C05482=1238.622,-59.773,-37.360,-179.966,5.213,148.890
C05483=1238.616,-59.523,-37.372,-179.963,5.213,148.889
C05484=1238.612,-59.273,-37.385,-179.961,5.213,148.889
C05485=1238.607,-59.024,-37.398,-179.958,5.213,148.888
C05486=1238.602,-58.774,-37.409,-179.956,5.214,148.887
C05487=1238.597,-58.525,-37.422,-179.953,5.214,148.887
C05488=1238.591,-58.275,-37.433,-179.951,5.214,148.886
C05489=1238.586,-58.026,-37.446,-179.949,5.214,148.885
C05490=1238.581,-57.777,-37.459,-179.946,5.214,148.884
C05491=1238.576,-57.526,-37.471,-179.943,5.214,148.884
C05492=1238.571,-57.277,-37.484,-179.941,5.214,148.883
C05493=1238.566,-57.027,-37.496,-179.939,5.214,148.882
C05494=1238.561,-56.777,-37.508,-179.936,5.214,148.881
C05495=1238.555,-56.528,-37.521,-179.934,5.214,148.881
C05496=1238.550,-56.279,-37.533,-179.931,5.214,148.880
C05497=1238.545,-56.028,-37.545,-179.929,5.214,148.879
C05498=1238.540,-55.779,-37.558,-179.927,5.215,148.879
C05499=1238.535,-55.529,-37.571,-179.924,5.214,148.878
C05500=1238.530,-55.280,-37.583,-179.922,5.215,148.877
C05501=1238.525,-55.030,-37.595,-179.920,5.214,148.877
C05502=1238.520,-54.780,-37.608,-179.917,5.215,148.876
C05503=1238.515,-54.530,-37.620,-179.914,5.215,148.875
C05504=1238.510,-54.281,-37.633,-179.912,5.215,148.874
C05505=1238.504,-54.032,-37.645,-179.909,5.215,148.873
C05506=1238.499,-53.782,-37.658,-179.907,5.215,148.873
C05507=1238.495,-53.532,-37.670,-179.904,5.215,148.872
C05508=1238.489,-53.282,-37.683,-179.902,5.215,148.871
C05509=1238.484,-53.033,-37.695,-179.900,5.216,148.871
C05510=1238.478,-52.783,-37.708,-179.898,5.215,148.870
C05511=1238.473,-52.533,-37.720,-179.895,5.216,148.869
C05512=1238.468,-52.283,-37.733,-179.893,5.215,148.869
C05513=1238.463,-52.034,-37.746,-179.890,5.216,148.868
C05514=1238.458,-51.785,-37.759,-179.888,5.216,148.867
C05515=1238.453,-51.536,-37.771,-179.885,5.216,148.866
C05516=1238.448,-51.285,-37.783,-179.882,5.216,148.865
C05517=1238.443,-51.036,-37.796,-179.880,5.216,148.865
C05518=1238.438,-50.786,-37.809,-179.877,5.216,148.864
C05519=1238.433,-50.537,-37.821,-179.875,5.216,148.863
C05520=1238.428,-50.287,-37.834,-179.873,5.217,148.863
C05521=1238.422,-50.037,-37.847,-179.871,5.216,148.862
C05522=1238.417,-49.788,-37.860,-179.868,5.217,148.861
C05523=1238.412,-49.538,-37.872,-179.866,5.216,148.861
C05524=1238.407,-49.288,-37.885,-179.863,5.217,148.860
C05525=1238.402,-49.039,-37.897,-179.861,5.217,148.859
C05526=1238.397,-48.789,-37.910,-179.858,5.217,148.858
C05527=1238.391,-48.519,-37.924,-179.855,5.217,148.858
C05528=1238.386,-48.250,-37.938,-179.853,5.217,148.857
C05529=1238.381,-47.981,-37.951,-179.850,5.217,148.856
C05530=1238.375,-47.711,-37.966,-179.847,5.217,148.855
C05531=1238.370,-47.461,-37.978,-179.845,5.217,148.854
C05532=1238.365,-47.212,-37.991,-179.843,5.218,148.854
C05533=1238.360,-46.962,-38.004,-179.840,5.217,148.853
C05534=1238.354,-46.712,-38.016,-179.838,5.218,148.852
C05535=1238.349,-46.462,-38.029,-179.836,5.218,148.852
C05536=1238.345,-46.212,-38.042,-179.833,5.218,148.851
C05537=1238.339,-45.963,-38.054,-179.830,5.219,148.850
C05538=1238.334,-45.714,-38.067,-179.828,5.218,148.850
C05539=1238.329,-45.463,-38.081,-179.826,5.219,148.849
C05540=1238.324,-45.214,-38.093,-179.823,5.218,148.848
C05541=1238.319,-44.965,-38.106,-179.820,5.219,148.847
C05542=1238.314,-44.715,-38.119,-179.818,5.218,148.847
C05543=1238.308,-44.465,-38.132,-179.816,5.219,148.846
C05544=1238.303,-44.216,-38.144,-179.814,5.218,148.845
C05545=1238.298,-43.966,-38.157,-179.811,5.219,148.844
C05546=1238.294,-43.716,-38.170,-179.808,5.219,148.844
C05547=1238.288,-43.467,-38.183,-179.806,5.219,148.843
C05548=1238.283,-43.217,-38.196,-179.803,5.220,148.842
C05549=1238.278,-42.967,-38.209,-179.801,5.219,148.842
C05550=1238.273,-42.719,-38.222,-179.799,5.220,148.841
C05551=1238.268,-42.468,-38.236,-179.796,5.219,148.840
C05552=1238.263,-42.219,-38.248,-179.793,5.220,148.839
C05553=1238.258,-41.970,-38.261,-179.791,5.219,148.839
C05554=1238.252,-41.719,-38.274,-179.789,5.220,148.838
C05555=1238.247,-41.470,-38.287,-179.786,5.220,148.837
C05556=1238.242,-41.221,-38.300,-179.784,5.220,148.836
C05557=1238.238,-40.971,-38.313,-179.781,5.220,148.836
C05558=1238.232,-40.721,-38.326,-179.779,5.220,148.835
C05559=1238.227,-40.471,-38.339,-179.777,5.221,148.834
C05560=1238.223,-40.222,-38.352,-179.774,5.220,148.834
C05561=1238.217,-39.973,-38.365,-179.772,5.221,148.833
C05562=1238.212,-39.723,-38.378,-179.769,5.221,148.832
C05563=1238.207,-39.473,-38.391,-179.767,5.221,148.831
C05564=1238.202,-39.223,-38.404,-179.764,5.221,148.831
C05565=1238.197,-38.974,-38.417,-179.762,5.221,148.830
C05566=1238.192,-38.725,-38.430,-179.759,5.221,148.829
C05567=1238.187,-38.475,-38.444,-179.757,5.221,148.829
C05568=1238.181,-38.225,-38.457,-179.754,5.222,148.828
C05569=1238.176,-37.975,-38.470,-179.752,5.222,148.827
C05570=1238.171,-37.726,-38.483,-179.750,5.222,148.826
C05571=1238.166,-37.477,-38.495,-179.747,5.222,148.826
C05572=1238.161,-37.227,-38.510,-179.745,5.222,148.825
C05573=1238.156,-36.977,-38.522,-179.742,5.222,148.824
C05574=1238.151,-36.727,-38.536,-179.740,5.222,148.824
C05575=1238.145,-36.478,-38.548,-179.737,5.222,148.823
C05576=1238.141,-36.228,-38.562,-179.734,5.223,148.822
C05577=1238.135,-35.979,-38.575,-179.732,5.222,148.821
C05578=1238.130,-35.729,-38.588,-179.730,5.223,148.821
C05579=1238.125,-35.479,-38.601,-179.728,5.223,148.820
C05580=1238.120,-35.230,-38.615,-179.725,5.223,148.819
C05581=1238.115,-34.980,-38.628,-179.722,5.224,148.819
C05582=1238.110,-34.731,-38.641,-179.720,5.223,148.818
C05583=1238.106,-34.481,-38.655,-179.717,5.224,148.817
C05584=1238.100,-34.232,-38.668,-179.715,5.224,148.816
C05585=1238.095,-33.982,-38.681,-179.713,5.224,148.816
C05586=1238.090,-33.733,-38.695,-179.711,5.224,148.815
C05587=1238.085,-33.483,-38.708,-179.707,5.224,148.814
C05588=1238.079,-33.233,-38.721,-179.705,5.224,148.813
C05589=1238.075,-32.984,-38.734,-179.703,5.224,148.813
C05590=1238.069,-32.734,-38.748,-179.700,5.225,148.812
C05591=1238.065,-32.484,-38.761,-179.698,5.224,148.811
C05592=1238.059,-32.235,-38.775,-179.695,5.225,148.811
C05593=1238.055,-31.985,-38.787,-179.693,5.225,148.810
C05594=1238.049,-31.735,-38.801,-179.691,5.225,148.809
C05595=1238.044,-31.486,-38.814,-179.688,5.226,148.809
C05596=1238.039,-31.236,-38.828,-179.686,5.225,148.808
C05597=1238.034,-30.987,-38.841,-179.683,5.226,148.807
C05598=1238.029,-30.737,-38.854,-179.681,5.225,148.806
C05599=1238.024,-30.487,-38.867,-179.678,5.226,148.805
C05600=1238.018,-30.238,-38.881,-179.675,5.226,148.805
C05601=1238.014,-29.988,-38.894,-179.673,5.226,148.804
C05602=1238.008,-29.739,-38.908,-179.671,5.226,148.803
C05603=1238.004,-29.489,-38.921,-179.668,5.226,148.803
C05604=1237.998,-29.240,-38.935,-179.666,5.227,148.802
C05605=1237.993,-28.990,-38.949,-179.663,5.227,148.801
C05606=1237.988,-28.741,-38.962,-179.661,5.227,148.801
C05607=1237.983,-28.491,-38.975,-179.658,5.227,148.800
C05608=1237.978,-28.242,-38.988,-179.656,5.227,148.799
C05609=1237.973,-27.992,-39.002,-179.654,5.227,148.798
C05610=1237.968,-27.742,-39.015,-179.651,5.228,148.798
C05611=1237.963,-27.493,-39.029,-179.649,5.228,148.797
C05612=1237.958,-27.243,-39.044,-179.646,5.228,148.796
C05613=1237.953,-26.994,-39.056,-179.644,5.228,148.795
C05614=1237.948,-26.744,-39.070,-179.641,5.228,148.795
C05615=1237.943,-26.495,-39.083,-179.638,5.229,148.794
C05616=1237.938,-26.245,-39.097,-179.636,5.228,148.793
C05617=1237.932,-25.995,-39.111,-179.634,5.229,148.793
C05618=1237.928,-25.746,-39.124,-179.631,5.228,148.792
C05619=1237.922,-25.496,-39.138,-179.629,5.229,148.791
C05620=1237.917,-25.247,-39.152,-179.626,5.229,148.791
C05621=1237.912,-24.997,-39.165,-179.624,5.229,148.790
C05622=1237.907,-24.747,-39.179,-179.621,5.230,148.789
C05623=1237.903,-24.498,-39.192,-179.619,5.229,148.789
C05624=1237.897,-24.248,-39.206,-179.616,5.230,148.788
C05625=1237.892,-23.999,-39.220,-179.614,5.230,148.787
C05626=1237.887,-23.749,-39.233,-179.611,5.230,148.786
C05627=1237.882,-23.499,-39.247,-179.609,5.230,148.785
C05628=1237.877,-23.250,-39.261,-179.606,5.231,148.785
C05629=1237.871,-23.000,-39.274,-179.604,5.230,148.784
C05630=1237.867,-22.750,-39.288,-179.601,5.231,148.783
C05631=1237.861,-22.482,-39.303,-179.599,5.232,148.783
C05632=1237.856,-22.212,-39.318,-179.596,5.231,148.782
C05633=1237.850,-21.943,-39.333,-179.593,5.231,148.781
C05634=1237.845,-21.674,-39.348,-179.591,5.232,148.780
C05635=1237.840,-21.425,-39.361,-179.589,5.232,148.780
C05636=1237.835,-21.174,-39.375,-179.586,5.232,148.779
C05637=1237.830,-20.925,-39.389,-179.583,5.232,148.778
C05638=1237.824,-20.676,-39.403,-179.581,5.232,148.777
C05639=1237.820,-20.426,-39.416,-179.578,5.232,148.777
C05640=1237.815,-20.176,-39.430,-179.576,5.232,148.776
C05641=1237.809,-19.927,-39.444,-179.573,5.233,148.775
C05642=1237.804,-19.677,-39.458,-179.571,5.233,148.775
C05643=1237.800,-19.427,-39.471,-179.569,5.233,148.774
C05644=1237.794,-19.178,-39.485,-179.566,5.233,148.773
C05645=1237.789,-18.929,-39.499,-179.563,5.234,148.773
C05646=1237.784,-18.679,-39.514,-179.561,5.234,148.772
C05647=1237.779,-18.430,-39.526,-179.559,5.234,148.771
C05648=1237.774,-18.180,-39.540,-179.557,5.234,148.770
C05649=1237.769,-17.930,-39.555,-179.554,5.234,148.770
C05650=1237.764,-17.681,-39.569,-179.551,5.235,148.769
C05651=1237.759,-17.431,-39.583,-179.549,5.234,148.768
C05652=1237.754,-17.181,-39.596,-179.546,5.235,148.767
C05653=1237.749,-16.932,-39.610,-179.543,5.235,148.767
C05654=1237.744,-16.683,-39.624,-179.541,5.235,148.766
C05655=1237.739,-16.433,-39.638,-179.539,5.236,148.765
C05656=1237.734,-16.183,-39.653,-179.537,5.235,148.765
C05657=1237.728,-15.934,-39.667,-179.534,5.236,148.764
C05658=1237.724,-15.685,-39.680,-179.531,5.236,148.763
C05659=1237.719,-15.435,-39.694,-179.529,5.236,148.763
C05660=1237.714,-15.185,-39.708,-179.526,5.237,148.762
C05661=1237.708,-14.936,-39.722,-179.524,5.237,148.761
C05662=1237.703,-14.686,-39.736,-179.522,5.237,148.760
C05663=1237.698,-14.436,-39.751,-179.519,5.237,148.760
C05664=1237.693,-14.187,-39.764,-179.516,5.237,148.759
C05665=1237.689,-13.938,-39.778,-179.514,5.237,148.758
C05666=1237.684,-13.688,-39.792,-179.511,5.238,148.757
C05667=1237.679,-13.439,-39.807,-179.509,5.237,148.757
C05668=1237.674,-13.189,-39.821,-179.506,5.238,148.756
C05669=1237.668,-12.939,-39.834,-179.504,5.238,148.755
C05670=1237.663,-12.689,-39.848,-179.502,5.238,148.755
C05671=1237.658,-12.440,-39.863,-179.499,5.239,148.754
C05672=1237.653,-12.190,-39.877,-179.496,5.239,148.753
C05673=1237.647,-11.941,-39.891,-179.494,5.239,148.753
C05674=1237.642,-11.691,-39.905,-179.492,5.239,148.752
C05675=1237.638,-11.442,-39.919,-179.489,5.240,148.751
C05676=1237.633,-11.192,-39.933,-179.487,5.240,148.751
C05677=1237.628,-10.943,-39.947,-179.484,5.240,148.750
C05678=1237.623,-10.694,-39.961,-179.482,5.241,148.749
C05679=1237.618,-10.444,-39.976,-179.479,5.240,148.748
C05680=1237.613,-10.194,-39.990,-179.476,5.241,148.748
C05681=1237.608,-9.944,-40.004,-179.474,5.241,148.747
C05682=1237.603,-9.695,-40.018,-179.472,5.241,148.746
C05683=1237.597,-9.446,-40.032,-179.469,5.241,148.745
C05684=1237.592,-9.196,-40.047,-179.467,5.241,148.745
C05685=1237.588,-8.947,-40.062,-179.464,5.242,148.744
C05686=1237.583,-8.697,-40.076,-179.462,5.242,148.743
C05687=1237.578,-8.447,-40.090,-179.460,5.242,148.743
C05688=1237.573,-8.198,-40.104,-179.457,5.242,148.742
C05689=1237.567,-7.949,-40.118,-179.454,5.243,148.741
C05690=1237.562,-7.699,-40.133,-179.452,5.243,148.741
C05691=1237.557,-7.449,-40.147,-179.449,5.243,148.740
C05692=1237.553,-7.200,-40.161,-179.447,5.244,148.739
C05693=1237.548,-6.950,-40.175,-179.445,5.243,148.739
C05694=1237.543,-6.700,-40.190,-179.442,5.244,148.738
C05695=1237.537,-6.452,-40.204,-179.439,5.244,148.737
C05696=1237.532,-6.202,-40.219,-179.437,5.244,148.736
C05697=1237.527,-5.952,-40.233,-179.434,5.244,148.736
C05698=1237.523,-5.703,-40.247,-179.432,5.245,148.735
C05699=1237.518,-5.453,-40.261,-179.429,5.245,148.734
C05700=1237.512,-5.203,-40.276,-179.427,5.245,148.733
C05701=1237.507,-4.954,-40.291,-179.424,5.246,148.733
C05702=1237.502,-4.704,-40.306,-179.422,5.245,148.732
C05703=1237.497,-4.455,-40.320,-179.419,5.246,148.731
C05704=1237.492,-4.205,-40.334,-179.417,5.246,148.731
C05705=1237.487,-3.956,-40.348,-179.415,5.246,148.730
C05706=1237.482,-3.707,-40.363,-179.412,5.247,148.729
C05707=1237.477,-3.457,-40.377,-179.409,5.247,148.729
C05708=1237.472,-3.207,-40.392,-179.407,5.247,148.728
C05709=1237.467,-2.957,-40.406,-179.405,5.247,148.727
C05710=1237.463,-2.708,-40.421,-179.402,5.248,148.727
C05711=1237.457,-2.458,-40.436,-179.399,5.247,148.726
C05712=1237.452,-2.209,-40.450,-179.397,5.248,148.725
C05713=1237.446,-1.960,-40.464,-179.394,5.248,148.724
C05714=1237.442,-1.711,-40.479,-179.392,5.248,148.724
C05715=1237.437,-1.461,-40.493,-179.389,5.249,148.723
C05716=1237.432,-1.211,-40.508,-179.387,5.249,148.722
C05717=1237.427,-0.961,-40.522,-179.385,5.249,148.721
C05718=1237.422,-0.712,-40.537,-179.382,5.249,148.721
C05719=1237.417,-0.462,-40.552,-179.379,5.250,148.720
C05720=1237.412,-0.213,-40.566,-179.377,5.251,148.719
C05721=1237.407,0.037,-40.581,-179.375,5.250,148.719
C05722=1237.402,0.286,-40.595,-179.372,5.251,148.718
C05723=1237.396,0.536,-40.610,-179.369,5.251,148.717
C05724=1237.392,0.785,-40.625,-179.367,5.251,148.717
C05725=1237.387,1.035,-40.639,-179.365,5.252,148.716
C05726=1237.382,1.284,-40.654,-179.362,5.252,148.715
C05727=1237.377,1.534,-40.669,-179.360,5.252,148.715
C05728=1237.371,1.784,-40.684,-179.357,5.252,148.714
C05729=1237.367,2.033,-40.698,-179.355,5.253,148.713
C05730=1237.362,2.283,-40.713,-179.352,5.252,148.712
C05731=1237.357,2.532,-40.728,-179.349,5.253,148.712
C05732=1237.351,2.782,-40.743,-179.347,5.253,148.711
C05733=1237.347,3.031,-40.757,-179.345,5.253,148.710
C05734=1237.342,3.281,-40.772,-179.342,5.254,148.710
C05735=1237.337,3.549,-40.788,-179.339,5.254,148.709
C05736=1237.330,3.818,-40.804,-179.337,5.255,148.708
C05737=1237.325,4.087,-40.819,-179.333,5.255,148.707
C05738=1237.320,4.355,-40.835,-179.331,5.255,148.707
C05739=1237.314,4.605,-40.850,-179.329,5.255,148.706
C05740=1237.310,4.854,-40.865,-179.326,5.256,148.705
C05741=1237.305,5.104,-40.879,-179.323,5.256,148.705
C05742=1237.299,5.354,-40.895,-179.321,5.256,148.704
C05743=1237.294,5.603,-40.909,-179.319,5.256,148.703
C05744=1237.290,5.853,-40.924,-179.316,5.257,148.702
C05745=1237.285,6.103,-40.939,-179.314,5.257,148.702
C05746=1237.280,6.352,-40.954,-179.311,5.257,148.701
C05747=1237.275,6.602,-40.968,-179.309,5.258,148.700
C05748=1237.270,6.851,-40.983,-179.307,5.258,148.700
C05749=1237.265,7.100,-40.999,-179.304,5.258,148.699
C05750=1237.260,7.350,-41.013,-179.301,5.259,148.698
C05751=1237.255,7.599,-41.028,-179.299,5.259,148.698
C05752=1237.250,7.849,-41.043,-179.297,5.259,148.697
C05753=1237.245,8.098,-41.058,-179.294,5.259,148.696
C05754=1237.240,8.348,-41.072,-179.291,5.260,148.695
C05755=1237.235,8.597,-41.088,-179.289,5.259,148.695
C05756=1237.230,8.847,-41.103,-179.286,5.260,148.694
C05757=1237.224,9.097,-41.118,-179.283,5.260,148.693
C05758=1237.220,9.346,-41.133,-179.281,5.261,148.693
C05759=1237.215,9.595,-41.148,-179.279,5.261,148.692
C05760=1237.209,9.845,-41.163,-179.276,5.261,148.691
C05761=1237.205,10.095,-41.178,-179.273,5.262,148.691
C05762=1237.200,10.345,-41.193,-179.271,5.262,148.690
C05763=1237.195,10.594,-41.208,-179.269,5.262,148.689
C05764=1237.190,10.843,-41.223,-179.266,5.263,148.688
C05765=1237.185,11.093,-41.238,-179.263,5.263,148.688
C05766=1237.180,11.342,-41.253,-179.261,5.263,148.687
C05767=1237.175,11.591,-41.268,-179.259,5.263,148.686
C05768=1237.170,11.840,-41.283,-179.256,5.264,148.686
C05769=1237.164,12.090,-41.298,-179.254,5.264,148.685
C05770=1237.160,12.340,-41.314,-179.251,5.264,148.684
C05771=1237.156,12.589,-41.329,-179.249,5.265,148.684
C05772=1237.150,12.839,-41.344,-179.246,5.265,148.683
C05773=1237.145,13.088,-41.359,-179.244,5.265,148.682
C05774=1237.140,13.338,-41.374,-179.241,5.266,148.682
C05775=1237.135,13.587,-41.389,-179.239,5.266,148.681
C05776=1237.130,13.837,-41.404,-179.236,5.267,148.680
C05777=1237.125,14.086,-41.419,-179.234,5.266,148.680
C05778=1237.120,14.336,-41.435,-179.231,5.267,148.679
C05779=1237.115,14.585,-41.450,-179.229,5.268,148.678
C05780=1237.110,14.835,-41.466,-179.226,5.267,148.678
C05781=1237.105,15.084,-41.480,-179.224,5.268,148.677
C05782=1237.100,15.334,-41.495,-179.221,5.268,148.676
C05783=1237.095,15.583,-41.510,-179.219,5.269,148.675
C05784=1237.090,15.833,-41.526,-179.216,5.269,148.675
C05785=1237.086,16.082,-41.541,-179.214,5.269,148.674
C05786=1237.080,16.332,-41.556,-179.211,5.270,148.673
C05787=1237.075,16.581,-41.571,-179.208,5.270,148.673
C05788=1237.070,16.830,-41.587,-179.206,5.270,148.672
C05789=1237.065,17.081,-41.603,-179.203,5.270,148.671
C05790=1237.060,17.330,-41.618,-179.201,5.271,148.670
C05791=1237.055,17.579,-41.633,-179.198,5.271,148.670
C05792=1237.050,17.828,-41.648,-179.196,5.271,148.669
C05793=1237.045,18.078,-41.664,-179.193,5.272,148.668
C05794=1237.041,18.328,-41.679,-179.191,5.272,148.668
C05795=1237.035,18.577,-41.694,-179.188,5.273,148.667
C05796=1237.030,18.827,-41.710,-179.186,5.272,148.666
C05797=1237.025,19.076,-41.725,-179.183,5.273,148.666
C05798=1237.020,19.325,-41.740,-179.181,5.274,148.665
C05799=1237.016,19.575,-41.756,-179.178,5.274,148.664
C05800=1237.010,19.824,-41.771,-179.176,5.274,148.664
C05801=1237.005,20.074,-41.787,-179.173,5.274,148.663
C05802=1237.000,20.323,-41.802,-179.171,5.275,148.662
C05803=1236.996,20.573,-41.818,-179.168,5.276,148.662
C05804=1236.990,20.822,-41.833,-179.166,5.275,148.661
C05805=1236.986,21.072,-41.848,-179.163,5.276,148.660
C05806=1236.980,21.321,-41.864,-179.161,5.276,148.660
C05807=1236.976,21.571,-41.879,-179.158,5.277,148.659
C05808=1236.971,21.820,-41.895,-179.156,5.277,148.658
C05809=1236.965,22.070,-41.910,-179.153,5.277,148.657
C05810=1236.961,22.319,-41.925,-179.151,5.278,148.657
C05811=1236.956,22.569,-41.941,-179.148,5.278,148.656
C05812=1236.951,22.818,-41.957,-179.146,5.278,148.655
C05813=1236.945,23.068,-41.973,-179.143,5.279,148.655
C05814=1236.941,23.317,-41.988,-179.141,5.279,148.654
C05815=1236.936,23.567,-42.004,-179.138,5.280,148.653
C05816=1236.930,23.816,-42.019,-179.136,5.279,148.653
C05817=1236.926,24.065,-42.034,-179.133,5.280,148.652
C05818=1236.921,24.315,-42.050,-179.131,5.281,148.651
C05819=1236.916,24.564,-42.066,-179.128,5.281,148.651
C05820=1236.911,24.813,-42.081,-179.125,5.282,148.650
C05821=1236.906,25.063,-42.097,-179.123,5.281,148.649
C05822=1236.901,25.313,-42.113,-179.121,5.282,148.649
C05823=1236.896,25.562,-42.128,-179.118,5.283,148.648
C05824=1236.891,25.811,-42.143,-179.115,5.283,148.647
C05825=1236.886,26.061,-42.159,-179.113,5.283,148.647
C05826=1236.881,26.311,-42.175,-179.111,5.283,148.646
C05827=1236.876,26.560,-42.191,-179.108,5.284,148.645
C05828=1236.872,26.809,-42.207,-179.105,5.285,148.645
C05829=1236.866,27.059,-42.222,-179.103,5.285,148.644
C05830=1236.861,27.308,-42.238,-179.100,5.285,148.643
C05831=1236.856,27.558,-42.254,-179.098,5.285,148.642
C05832=1236.851,27.807,-42.270,-179.095,5.286,148.642
C05833=1236.846,28.056,-42.285,-179.093,5.286,148.641
C05834=1236.842,28.306,-42.301,-179.090,5.286,148.640
C05835=1236.836,28.556,-42.317,-179.088,5.287,148.640
C05836=1236.831,28.806,-42.333,-179.085,5.287,148.639
C05837=1236.826,29.054,-42.349,-179.083,5.288,148.638
C05838=1236.822,29.304,-42.364,-179.080,5.288,148.638
C05839=1236.816,29.572,-42.381,-179.078,5.288,148.637
C05840=1236.811,29.841,-42.398,-179.075,5.289,148.636
C05841=1236.806,30.110,-42.415,-179.073,5.289,148.636
C05842=1236.800,30.378,-42.432,-179.069,5.290,148.635
C05843=1236.795,30.628,-42.448,-179.067,5.290,148.634
C05844=1236.790,30.877,-42.465,-179.064,5.291,148.633
C05845=1236.785,31.126,-42.480,-179.061,5.291,148.633
C05846=1236.781,31.376,-42.496,-179.059,5.291,148.632
C05847=1236.775,31.626,-42.511,-179.057,5.292,148.631
C05848=1236.771,31.875,-42.528,-179.054,5.292,148.631
C05849=1236.765,32.125,-42.543,-179.051,5.293,148.630
C05850=1236.760,32.374,-42.559,-179.049,5.293,148.629
C05851=1236.756,32.623,-42.576,-179.047,5.293,148.629
C05852=1236.750,32.873,-42.591,-179.045,5.294,148.628
C05853=1236.746,33.122,-42.608,-179.042,5.294,148.628
C05854=1236.740,33.372,-42.623,-179.039,5.295,148.627
C05855=1236.735,33.621,-42.639,-179.037,5.296,148.626
C05856=1236.731,33.870,-42.655,-179.035,5.295,148.626
C05857=1236.726,34.120,-42.671,-179.032,5.296,148.625
C05858=1236.721,34.369,-42.687,-179.029,5.296,148.624
C05859=1236.716,34.619,-42.703,-179.027,5.297,148.623
C05860=1236.711,34.869,-42.719,-179.024,5.298,148.623
C05861=1236.706,35.117,-42.735,-179.022,5.297,148.622
C05862=1236.701,35.368,-42.751,-179.019,5.298,148.621
C05863=1236.696,35.616,-42.768,-179.017,5.298,148.621
C05864=1236.691,35.866,-42.783,-179.014,5.299,148.620
C05865=1236.686,36.115,-42.800,-179.011,5.300,148.619
C05866=1236.681,36.365,-42.815,-179.009,5.300,148.619
C05867=1236.677,36.614,-42.832,-179.007,5.300,148.618
C05868=1236.671,36.864,-42.848,-179.004,5.300,148.617
C05869=1236.667,37.113,-42.864,-179.001,5.301,148.617
C05870=1236.661,37.362,-42.880,-178.999,5.302,148.616
C05871=1236.657,37.612,-42.897,-178.996,5.302,148.615
C05872=1236.651,37.861,-42.912,-178.994,5.302,148.615
C05873=1236.647,38.111,-42.929,-178.991,5.303,148.614
C05874=1236.642,38.360,-42.944,-178.989,5.303,148.613
C05875=1236.637,38.610,-42.961,-178.986,5.304,148.613
C05876=1236.632,38.859,-42.977,-178.983,5.304,148.612
C05877=1236.627,39.109,-42.993,-178.981,5.305,148.611
C05878=1236.622,39.358,-43.009,-178.979,5.305,148.611
C05879=1236.617,39.607,-43.026,-178.976,5.305,148.610
C05880=1236.612,39.856,-43.042,-178.974,5.306,148.609
C05881=1236.607,40.107,-43.058,-178.971,5.306,148.609
C05882=1236.602,40.355,-43.075,-178.968,5.307,148.608
C05883=1236.597,40.606,-43.091,-178.966,5.307,148.607
C05884=1236.592,40.854,-43.107,-178.964,5.307,148.607
C05885=1236.587,41.104,-43.124,-178.961,5.308,148.606
C05886=1236.583,41.354,-43.140,-178.959,5.309,148.605
C05887=1236.577,41.603,-43.156,-178.956,5.309,148.605
C05888=1236.573,41.852,-43.173,-178.953,5.310,148.604
C05889=1236.568,42.102,-43.188,-178.951,5.310,148.603
C05890=1236.563,42.351,-43.205,-178.949,5.310,148.603
C05891=1236.557,42.600,-43.222,-178.946,5.311,148.602
C05892=1236.552,42.850,-43.238,-178.943,5.311,148.601
C05893=1236.547,43.099,-43.254,-178.941,5.312,148.601
C05894=1236.543,43.349,-43.271,-178.938,5.312,148.600
C05895=1236.538,43.599,-43.287,-178.936,5.313,148.599
C05896=1236.533,43.847,-43.303,-178.933,5.313,148.599
C05897=1236.529,44.097,-43.320,-178.931,5.313,148.598
C05898=1236.523,44.346,-43.336,-178.928,5.314,148.597
C05899=1236.518,44.596,-43.352,-178.926,5.314,148.597
C05900=1236.513,44.845,-43.369,-178.923,5.315,148.596
C05901=1236.508,45.094,-43.385,-178.920,5.316,148.595
C05902=1236.504,45.344,-43.402,-178.918,5.316,148.595
C05903=1236.498,45.594,-43.418,-178.916,5.316,148.594
C05904=1236.493,45.843,-43.435,-178.913,5.317,148.594
C05905=1236.489,46.093,-43.452,-178.911,5.317,148.593
C05906=1236.484,46.341,-43.468,-178.908,5.318,148.592
C05907=1236.479,46.591,-43.485,-178.906,5.319,148.592
C05908=1236.473,46.841,-43.501,-178.903,5.319,148.591
C05909=1236.469,47.090,-43.517,-178.900,5.320,148.590
C05910=1236.464,47.340,-43.534,-178.898,5.319,148.590
C05911=1236.459,47.588,-43.550,-178.896,5.320,148.589
C05912=1236.454,47.838,-43.568,-178.893,5.321,148.588
C05913=1236.449,48.088,-43.584,-178.890,5.321,148.588
C05914=1236.444,48.337,-43.600,-178.888,5.322,148.587
C05915=1236.440,48.586,-43.617,-178.885,5.322,148.586
C05916=1236.434,48.836,-43.634,-178.882,5.323,148.586
C05917=1236.429,49.085,-43.650,-178.880,5.323,148.585
C05918=1236.425,49.335,-43.667,-178.878,5.323,148.584
C05919=1236.420,49.584,-43.683,-178.876,5.324,148.584
C05920=1236.414,49.833,-43.700,-178.873,5.325,148.583
C05921=1236.410,50.083,-43.717,-178.870,5.325,148.582
C05922=1236.406,50.332,-43.734,-178.868,5.326,148.582
C05923=1236.400,50.581,-43.751,-178.865,5.327,148.581
C05924=1236.395,50.831,-43.767,-178.862,5.327,148.580
C05925=1236.390,51.081,-43.783,-178.860,5.327,148.580
C05926=1236.385,51.330,-43.800,-178.858,5.327,148.579
C05927=1236.380,51.579,-43.817,-178.855,5.328,148.578
C05928=1236.376,51.829,-43.833,-178.852,5.329,148.578
C05929=1236.370,52.078,-43.850,-178.850,5.329,148.577
C05930=1236.365,52.327,-43.867,-178.847,5.330,148.576
C05931=1236.361,52.577,-43.884,-178.844,5.330,148.576
C05932=1236.356,52.827,-43.901,-178.842,5.331,148.575
C05933=1236.351,53.075,-43.917,-178.840,5.331,148.575
C05934=1236.346,53.325,-43.934,-178.838,5.332,148.574
C05935=1236.341,53.575,-43.951,-178.835,5.332,148.573
C05936=1236.336,53.824,-43.968,-178.832,5.333,148.573
C05937=1236.332,54.072,-43.985,-178.830,5.333,148.572
C05938=1236.326,54.322,-44.002,-178.827,5.334,148.571
C05939=1236.322,54.572,-44.019,-178.824,5.335,148.571
C05940=1236.316,54.821,-44.036,-178.822,5.335,148.570
C05941=1236.312,55.070,-44.052,-178.819,5.336,148.569
C05942=1236.307,55.320,-44.069,-178.817,5.335,148.569
C05943=1236.301,55.588,-44.087,-178.814,5.336,148.568
C05944=1236.296,55.856,-44.106,-178.811,5.337,148.567
C05945=1236.291,56.125,-44.124,-178.809,5.338,148.567
C05946=1236.286,56.393,-44.142,-178.806,5.339,148.566
C05947=1236.281,56.643,-44.159,-178.803,5.339,148.565
C05948=1236.276,56.892,-44.176,-178.801,5.339,148.565
C05949=1236.270,57.142,-44.193,-178.799,5.340,148.564
C05950=1236.266,57.391,-44.209,-178.796,5.340,148.563
C05951=1236.261,57.640,-44.227,-178.793,5.341,148.563
C05952=1236.256,57.890,-44.244,-178.791,5.341,148.562
C05953=1236.251,58.139,-44.261,-178.789,5.342,148.561
C05954=1236.246,58.388,-44.278,-178.786,5.343,148.561
C05955=1236.241,58.638,-44.295,-178.783,5.343,148.560
C05956=1236.237,58.887,-44.312,-178.781,5.344,148.559
C05957=1236.232,59.137,-44.330,-178.778,5.345,148.559
C05958=1236.227,59.386,-44.346,-178.776,5.344,148.558
C05959=1236.221,59.635,-44.363,-178.773,5.345,148.557
C05960=1236.217,59.885,-44.380,-178.771,5.346,148.557
C05961=1236.212,60.134,-44.398,-178.768,5.346,148.556
C05962=1236.207,60.383,-44.414,-178.765,5.347,148.555
C05963=1236.202,60.633,-44.432,-178.763,5.348,148.555
C05964=1236.197,60.881,-44.449,-178.761,5.348,148.554
C05965=1236.192,61.131,-44.466,-178.758,5.349,148.554
C05966=1236.187,61.381,-44.483,-178.755,5.349,148.553
C05967=1236.182,61.630,-44.500,-178.753,5.350,148.552
C05968=1236.178,61.880,-44.518,-178.750,5.351,148.552
C05969=1236.173,62.129,-44.535,-178.748,5.351,148.551
C05970=1236.168,62.379,-44.552,-178.745,5.352,148.550
C05971=1236.163,62.627,-44.569,-178.743,5.352,148.550
C05972=1236.158,62.877,-44.586,-178.741,5.352,148.549
C05973=1236.153,63.127,-44.603,-178.738,5.353,148.549
C05974=1236.148,63.376,-44.621,-178.735,5.354,148.548
C05975=1236.143,63.625,-44.638,-178.733,5.354,148.547
C05976=1236.139,63.874,-44.655,-178.730,5.355,148.547
C05977=1236.134,64.124,-44.673,-178.728,5.355,148.546
C05978=1236.129,64.374,-44.690,-178.725,5.356,148.545
C05979=1236.124,64.622,-44.707,-178.722,5.357,148.545
C05980=1236.119,64.872,-44.724,-178.720,5.358,148.544
C05981=1236.114,65.121,-44.742,-178.717,5.358,148.543
C05982=1236.109,65.370,-44.759,-178.715,5.359,148.543
C05983=1236.104,65.620,-44.776,-178.712,5.359,148.542
C05984=1236.099,65.869,-44.794,-178.710,5.360,148.541
C05985=1236.095,66.119,-44.811,-178.707,5.360,148.541
C05986=1236.090,66.368,-44.829,-178.705,5.360,148.540
C05987=1236.085,66.618,-44.846,-178.702,5.361,148.539
C05988=1236.080,66.867,-44.863,-178.700,5.362,148.539
C05989=1236.075,67.117,-44.881,-178.698,5.362,148.538
C05990=1236.070,67.365,-44.898,-178.695,5.363,148.538
C05991=1236.065,67.614,-44.915,-178.692,5.364,148.537
C05992=1236.060,67.864,-44.933,-178.690,5.364,148.536
C05993=1236.055,68.113,-44.950,-178.687,5.365,148.536
C05994=1236.051,68.362,-44.968,-178.684,5.365,148.535
C05995=1236.046,68.612,-44.985,-178.682,5.366,148.535
C05996=1236.041,68.861,-45.003,-178.680,5.367,148.534
C05997=1236.035,69.111,-45.020,-178.677,5.367,148.533
C05998=1236.031,69.360,-45.038,-178.674,5.368,148.533
C05999=1236.026,69.609,-45.055,-178.672,5.369,148.532
C06000=1236.021,69.859,-45.073,-178.669,5.369,148.531
C06001=1236.016,70.108,-45.091,-178.666,5.370,148.531
C06002=1236.012,70.358,-45.107,-178.664,5.371,148.530
C06003=1236.007,70.607,-45.125,-178.662,5.371,148.530
C06004=1236.002,70.856,-45.143,-178.659,5.372,148.529
C06005=1235.997,71.106,-45.161,-178.656,5.373,148.528
C06006=1235.993,71.355,-45.178,-178.654,5.373,148.528
C06007=1235.987,71.604,-45.195,-178.651,5.374,148.527
C06008=1235.982,71.854,-45.213,-178.649,5.374,148.526
C06009=1235.978,72.103,-45.231,-178.647,5.375,148.526
C06010=1235.972,72.353,-45.248,-178.644,5.375,148.525
C06011=1235.967,72.602,-45.266,-178.642,5.376,148.525
C06012=1235.963,72.851,-45.284,-178.639,5.376,148.524
C06013=1235.958,73.100,-45.301,-178.636,5.377,148.523
C06014=1235.953,73.350,-45.319,-178.634,5.377,148.523
C06015=1235.948,73.599,-45.337,-178.632,5.378,148.522
C06016=1235.943,73.848,-45.355,-178.629,5.379,148.521
C06017=1235.938,74.098,-45.372,-178.626,5.380,148.521
C06018=1235.934,74.347,-45.390,-178.624,5.380,148.520
C06019=1235.929,74.596,-45.408,-178.621,5.381,148.519
C06020=1235.924,74.846,-45.425,-178.619,5.381,148.519
C06021=1235.919,75.095,-45.443,-178.616,5.382,148.518
C06022=1235.914,75.344,-45.461,-178.614,5.383,148.518
C06023=1235.909,75.593,-45.479,-178.611,5.384,148.517
C06024=1235.904,75.842,-45.497,-178.609,5.384,148.516
C06025=1235.899,76.092,-45.514,-178.606,5.385,148.516
C06026=1235.894,76.341,-45.532,-178.603,5.385,148.515
C06027=1235.890,76.591,-45.550,-178.601,5.386,148.515
C06028=1235.886,76.840,-45.568,-178.599,5.387,148.514
C06029=1235.881,77.089,-45.586,-178.596,5.388,148.513
C06030=1235.875,77.339,-45.603,-178.593,5.388,148.513
C06031=1235.870,77.588,-45.621,-178.591,5.389,148.512
C06032=1235.866,77.837,-45.639,-178.588,5.389,148.511
C06033=1235.861,78.086,-45.657,-178.586,5.390,148.511
C06034=1235.856,78.336,-45.675,-178.583,5.391,148.510
C06035=1235.851,78.585,-45.693,-178.581,5.391,148.510
C06036=1235.846,78.834,-45.711,-178.578,5.392,148.509
C06037=1235.841,79.083,-45.729,-178.575,5.393,148.508
C06038=1235.836,79.334,-45.747,-178.573,5.394,148.508
C06039=1235.831,79.583,-45.765,-178.571,5.394,148.507
C06040=1235.827,79.832,-45.783,-178.568,5.395,148.507
C06041=1235.822,80.081,-45.801,-178.565,5.395,148.506
C06042=1235.817,80.330,-45.819,-178.563,5.396,148.505
C06043=1235.812,80.579,-45.836,-178.560,5.397,148.505
C06044=1235.807,80.829,-45.854,-178.558,5.398,148.504
C06045=1235.802,81.078,-45.872,-178.555,5.398,148.504
C06046=1235.798,81.328,-45.891,-178.553,5.399,148.503
C06047=1235.793,81.596,-45.910,-178.550,5.399,148.502
C06048=1235.788,81.864,-45.930,-178.547,5.401,148.502
C06049=1235.782,82.132,-45.949,-178.544,5.401,148.501
C06050=1235.777,82.401,-45.969,-178.542,5.402,148.500
C06051=1235.772,82.650,-45.987,-178.539,5.403,148.500
C06052=1235.767,82.899,-46.005,-178.536,5.403,148.499
C06053=1235.762,83.149,-46.023,-178.534,5.404,148.499
C06054=1235.757,83.398,-46.041,-178.532,5.405,148.498
C06055=1235.753,83.648,-46.059,-178.529,5.405,148.497
C06056=1235.748,83.897,-46.077,-178.526,5.406,148.497
C06057=1235.743,84.146,-46.095,-178.524,5.407,148.496
C06058=1235.738,84.395,-46.113,-178.522,5.408,148.495
C06059=1235.733,84.644,-46.131,-178.519,5.408,148.495
C06060=1235.728,84.893,-46.149,-178.516,5.409,148.494
C06061=1235.723,85.144,-46.168,-178.514,5.409,148.493
C06062=1235.718,85.393,-46.186,-178.511,5.410,148.493
C06063=1235.713,85.642,-46.204,-178.509,5.411,148.492
C06064=1235.709,85.891,-46.223,-178.506,5.412,148.492
C06065=1235.704,86.140,-46.241,-178.504,5.412,148.491
C06066=1235.699,86.390,-46.259,-178.501,5.413,148.490
C06067=1235.694,86.639,-46.277,-178.499,5.413,148.490
C06068=1235.689,86.888,-46.296,-178.496,5.414,148.489
C06069=1235.684,87.137,-46.314,-178.494,5.415,148.489
C06070=1235.680,87.387,-46.332,-178.491,5.416,148.488
C06071=1235.675,87.636,-46.351,-178.488,5.417,148.487
C06072=1235.670,87.885,-46.369,-178.486,5.418,148.487
C06073=1235.665,88.134,-46.387,-178.483,5.419,148.486
C06074=1235.660,88.384,-46.406,-178.481,5.419,148.486
C06075=1235.655,88.634,-46.424,-178.478,5.420,148.485
C06076=1235.651,88.882,-46.442,-178.475,5.420,148.484
C06077=1235.646,89.131,-46.460,-178.473,5.421,148.484
C06078=1235.641,89.381,-46.479,-178.471,5.422,148.483
C06079=1235.636,89.631,-46.497,-178.468,5.423,148.483
C06080=1235.631,89.879,-46.516,-178.465,5.423,148.482
C06081=1235.626,90.128,-46.534,-178.463,5.424,148.482
C06082=1235.622,90.378,-46.552,-178.461,5.425,148.481
C06083=1235.617,90.627,-46.571,-178.458,5.425,148.480
C06084=1235.612,90.876,-46.589,-178.455,5.426,148.480
C06085=1235.607,91.126,-46.608,-178.453,5.427,148.479
C06086=1235.602,91.375,-46.626,-178.451,5.428,148.479
C06087=1235.597,91.624,-46.645,-178.448,5.428,148.478
C06088=1235.593,91.874,-46.663,-178.445,5.430,148.477
C06089=1235.588,92.123,-46.682,-178.442,5.430,148.477
C06090=1235.583,92.372,-46.701,-178.440,5.431,148.476
C06091=1235.578,92.621,-46.719,-178.437,5.432,148.476
C06092=1235.574,92.871,-46.738,-178.435,5.432,148.475
C06093=1235.568,93.120,-46.756,-178.432,5.433,148.474
C06094=1235.563,93.369,-46.774,-178.430,5.434,148.474
C06095=1235.559,93.619,-46.793,-178.427,5.435,148.473
C06096=1235.554,93.868,-46.811,-178.425,5.435,148.473
C06097=1235.549,94.117,-46.831,-178.422,5.436,148.472
C06098=1235.544,94.367,-46.849,-178.420,5.437,148.471
C06099=1235.540,94.616,-46.867,-178.418,5.437,148.471
C06100=1235.534,94.865,-46.886,-178.415,5.438,148.470
C06101=1235.530,95.114,-46.905,-178.412,5.440,148.469
C06102=1235.525,95.363,-46.924,-178.410,5.440,148.469
C06103=1235.520,95.613,-46.942,-178.407,5.441,148.468
C06104=1235.516,95.862,-46.961,-178.404,5.442,148.468
C06105=1235.510,96.111,-46.979,-178.402,5.442,148.467
C06106=1235.506,96.360,-46.999,-178.400,5.443,148.467
C06107=1235.501,96.610,-47.017,-178.397,5.444,148.466
C06108=1235.496,96.858,-47.036,-178.394,5.445,148.465
C06109=1235.491,97.108,-47.054,-178.392,5.445,148.465
C06110=1235.486,97.357,-47.073,-178.390,5.446,148.464
C06111=1235.482,97.607,-47.092,-178.387,5.447,148.464
C06112=1235.476,97.856,-47.111,-178.384,5.448,148.463
C06113=1235.472,98.105,-47.129,-178.382,5.449,148.463
C06114=1235.467,98.354,-47.148,-178.379,5.450,148.462
C06115=1235.462,98.603,-47.167,-178.376,5.450,148.461
C06116=1235.458,98.853,-47.186,-178.374,5.451,148.461
C06117=1235.452,99.102,-47.205,-178.372,5.452,148.460
C06118=1235.448,99.351,-47.223,-178.369,5.453,148.460
C06119=1235.443,99.601,-47.243,-178.366,5.453,148.459
C06120=1235.438,99.850,-47.261,-178.364,5.454,148.458
C06121=1235.433,100.100,-47.280,-178.362,5.455,148.458
C06122=1235.429,100.348,-47.299,-178.359,5.456,148.457
C06123=1235.424,100.598,-47.318,-178.356,5.457,148.457
C06124=1235.419,100.847,-47.337,-178.354,5.458,148.456
C06125=1235.414,101.096,-47.356,-178.351,5.458,148.456
C06126=1235.409,101.346,-47.374,-178.349,5.459,148.455
C06127=1235.404,101.594,-47.394,-178.346,5.460,148.454
C06128=1235.400,101.844,-47.413,-178.344,5.461,148.454
C06129=1235.394,102.093,-47.431,-178.341,5.461,148.453
C06130=1235.390,102.342,-47.450,-178.339,5.462,148.453
C06131=1235.385,102.591,-47.470,-178.336,5.464,148.452
C06132=1235.381,102.841,-47.489,-178.333,5.464,148.452
C06133=1235.375,103.090,-47.507,-178.331,5.465,148.451
C06134=1235.371,103.339,-47.526,-178.328,5.466,148.450
C06135=1235.366,103.588,-47.546,-178.326,5.467,148.450
C06136=1235.361,103.838,-47.565,-178.323,5.467,148.449
C06137=1235.356,104.087,-47.583,-178.321,5.468,148.448
C06138=1235.352,104.336,-47.603,-178.319,5.469,148.448
C06139=1235.347,104.585,-47.622,-178.315,5.470,148.447
C06140=1235.342,104.835,-47.641,-178.313,5.471,148.447
C06141=1235.337,105.084,-47.660,-178.310,5.471,148.446
C06142=1235.333,105.333,-47.679,-178.308,5.472,148.446
C06143=1235.327,105.582,-47.698,-178.305,5.473,148.445
C06144=1235.323,105.831,-47.717,-178.303,5.474,148.444
C06145=1235.318,106.080,-47.736,-178.301,5.475,148.444
C06146=1235.313,106.330,-47.756,-178.298,5.476,148.443
C06147=1235.308,106.579,-47.774,-178.295,5.477,148.443
C06148=1235.303,106.829,-47.794,-178.293,5.478,148.442
C06149=1235.298,107.078,-47.813,-178.290,5.478,148.442
C06150=1235.294,107.327,-47.832,-178.288,5.479,148.441
C06151=1235.289,107.595,-47.853,-178.285,5.480,148.440
C06152=1235.284,107.863,-47.874,-178.282,5.481,148.440
C06153=1235.278,108.133,-47.894,-178.280,5.482,148.439
C06154=1235.273,108.401,-47.915,-178.277,5.483,148.439
C06155=1235.268,108.650,-47.935,-178.274,5.484,148.438
C06156=1235.264,108.899,-47.953,-178.271,5.485,148.437
C06157=1235.259,109.148,-47.973,-178.269,5.486,148.437
C06158=1235.254,109.398,-47.993,-178.267,5.486,148.436
C06159=1235.249,109.646,-48.011,-178.264,5.487,148.436
C06160=1235.245,109.896,-48.031,-178.262,5.488,148.435
C06161=1235.239,110.145,-48.050,-178.259,5.489,148.435
C06162=1235.235,110.394,-48.070,-178.256,5.490,148.434
C06163=1235.230,110.643,-48.089,-178.254,5.491,148.434
C06164=1235.225,110.893,-48.108,-178.251,5.492,148.433
C06165=1235.221,111.142,-48.128,-178.249,5.492,148.432
C06166=1235.215,111.391,-48.147,-178.247,5.493,148.432
C06167=1235.211,111.640,-48.166,-178.244,5.494,148.431
C06168=1235.206,111.890,-48.186,-178.241,5.495,148.431
C06169=1235.201,112.139,-48.205,-178.239,5.496,148.430
C06170=1235.196,112.388,-48.225,-178.236,5.497,148.430
C06171=1235.192,112.637,-48.244,-178.233,5.497,148.429
C06172=1235.187,112.886,-48.263,-178.231,5.498,148.429
C06173=1235.182,113.136,-48.283,-178.228,5.500,148.428
C06174=1235.177,113.385,-48.302,-178.226,5.501,148.427
C06175=1235.172,113.634,-48.323,-178.223,5.502,148.427
C06176=1235.168,113.883,-48.342,-178.221,5.502,148.426
C06177=1235.163,114.132,-48.361,-178.218,5.503,148.426
C06178=1235.158,114.381,-48.381,-178.216,5.504,148.425
C06179=1235.154,114.631,-48.400,-178.213,5.505,148.425
C06180=1235.148,114.880,-48.420,-178.210,5.506,148.424
C06181=1235.144,115.129,-48.439,-178.208,5.507,148.424
C06182=1235.139,115.378,-48.460,-178.206,5.507,148.423
C06183=1235.135,115.627,-48.478,-178.203,5.508,148.422
C06184=1235.130,115.877,-48.498,-178.200,5.510,148.422
C06185=1235.125,116.126,-48.518,-178.198,5.511,148.421
C06186=1235.120,116.375,-48.537,-178.195,5.511,148.421
C06187=1235.115,116.624,-48.557,-178.193,5.512,148.420
C06188=1235.111,116.873,-48.577,-178.190,5.513,148.420
C06189=1235.105,117.122,-48.596,-178.188,5.515,148.419
C06190=1235.100,117.372,-48.616,-178.185,5.515,148.418
C06191=1235.096,117.621,-48.636,-178.182,5.516,148.418
C06192=1235.091,117.869,-48.655,-178.180,5.517,148.417
C06193=1235.087,118.119,-48.675,-178.178,5.517,148.417
C06194=1235.082,118.369,-48.694,-178.175,5.519,148.416
C06195=1235.077,118.617,-48.715,-178.172,5.520,148.416
C06196=1235.072,118.866,-48.734,-178.170,5.521,148.415
C06197=1235.067,119.116,-48.754,-178.167,5.521,148.414
C06198=1235.063,119.366,-48.773,-178.165,5.522,148.414
C06199=1235.058,119.614,-48.794,-178.162,5.524,148.413
C06200=1235.053,119.863,-48.813,-178.160,5.525,148.413
C06201=1235.048,120.113,-48.833,-178.157,5.525,148.412
C06202=1235.044,120.362,-48.853,-178.155,5.526,148.412
C06203=1235.038,120.611,-48.872,-178.152,5.527,148.411
C06204=1235.034,120.860,-48.893,-178.149,5.528,148.411
C06205=1235.029,121.109,-48.912,-178.147,5.529,148.410
C06206=1235.024,121.359,-48.932,-178.145,5.530,148.410
C06207=1235.020,121.608,-48.952,-178.142,5.531,148.409
C06208=1235.015,121.857,-48.972,-178.139,5.532,148.409
C06209=1235.010,122.106,-48.992,-178.137,5.533,148.408
C06210=1235.005,122.355,-49.012,-178.134,5.534,148.407
C06211=1235.001,122.605,-49.031,-178.132,5.535,148.407
C06212=1234.996,122.853,-49.051,-178.129,5.535,148.406
C06213=1234.991,123.102,-49.071,-178.127,5.537,148.406
C06214=1234.986,123.351,-49.091,-178.124,5.538,148.405
C06215=1234.982,123.601,-49.111,-178.121,5.538,148.405
C06216=1234.977,123.850,-49.131,-178.119,5.539,148.404
C06217=1234.972,124.099,-49.151,-178.116,5.541,148.404
C06218=1234.968,124.348,-49.171,-178.114,5.542,148.403
C06219=1234.962,124.598,-49.191,-178.111,5.542,148.403
C06220=1234.958,124.847,-49.212,-178.109,5.543,148.402
C06221=1234.953,125.096,-49.231,-178.106,5.545,148.402
C06222=1234.948,125.345,-49.252,-178.104,5.546,148.401
C06223=1234.943,125.594,-49.271,-178.101,5.546,148.401
C06224=1234.939,125.843,-49.291,-178.099,5.547,148.400
C06225=1234.934,126.093,-49.311,-178.096,5.549,148.399
C06226=1234.929,126.341,-49.331,-178.094,5.550,148.399
C06227=1234.925,126.590,-49.352,-178.091,5.550,148.398
C06228=1234.920,126.840,-49.372,-178.089,5.551,148.398
C06229=1234.915,127.089,-49.392,-178.086,5.553,148.397
C06230=1234.910,127.338,-49.412,-178.083,5.553,148.397
C06231=1234.905,127.587,-49.432,-178.081,5.554,148.396
C06232=1234.901,127.836,-49.452,-178.078,5.555,148.396
C06233=1234.896,128.086,-49.472,-178.076,5.557,148.395
C06234=1234.891,128.335,-49.493,-178.073,5.557,148.395
C06235=1234.887,128.584,-49.513,-178.071,5.558,148.394
C06236=1234.882,128.833,-49.533,-178.068,5.559,148.393
C06237=1234.877,129.082,-49.553,-178.065,5.560,148.393
C06238=1234.872,129.331,-49.573,-178.063,5.561,148.392
C06239=1234.867,129.580,-49.594,-178.060,5.562,148.392
C06240=1234.862,129.829,-49.614,-178.058,5.564,148.391
C06241=1234.858,130.078,-49.634,-178.055,5.565,148.391
C06242=1234.853,130.328,-49.654,-178.053,5.565,148.390
C06243=1234.849,130.577,-49.674,-178.050,5.566,148.390
C06244=1234.844,130.826,-49.695,-178.047,5.568,148.389
C06245=1234.839,131.075,-49.716,-178.045,5.569,148.389
C06246=1234.834,131.325,-49.735,-178.043,5.569,148.388
C06247=1234.829,131.574,-49.756,-178.040,5.570,148.388
C06248=1234.825,131.823,-49.777,-178.037,5.572,148.387
C06249=1234.820,132.071,-49.797,-178.035,5.573,148.387
C06250=1234.815,132.321,-49.816,-178.033,5.573,148.386
C06251=1234.810,132.570,-49.837,-178.029,5.575,148.385
C06252=1234.805,132.819,-49.858,-178.027,5.576,148.385
C06253=1234.801,133.068,-49.878,-178.025,5.577,148.384
C06254=1234.796,133.317,-49.899,-178.023,5.577,148.384
C06255=1234.791,133.586,-49.920,-178.019,5.579,148.383
C06256=1234.786,133.855,-49.943,-178.017,5.580,148.383
C06257=1234.781,134.123,-49.965,-178.014,5.581,148.382
C06258=1234.775,134.392,-49.987,-178.012,5.582,148.382
C06259=1234.771,134.641,-50.007,-178.008,5.584,148.381
C06260=1234.766,134.890,-50.028,-178.006,5.585,148.381
C06261=1234.761,135.139,-50.049,-178.004,5.585,148.380
C06262=1234.757,135.388,-50.069,-178.001,5.587,148.380
C06263=1234.752,135.637,-50.089,-177.998,5.588,148.379
C06264=1234.747,135.886,-50.110,-177.996,5.588,148.378
C06265=1234.742,136.136,-50.130,-177.994,5.589,148.378
C06266=1234.738,136.385,-50.150,-177.991,5.591,148.377
C06267=1234.733,136.634,-50.171,-177.988,5.592,148.377
C06268=1234.728,136.883,-50.192,-177.986,5.592,148.376
C06269=1234.723,137.132,-50.213,-177.983,5.594,148.376
C06270=1234.719,137.381,-50.233,-177.981,5.595,148.375
C06271=1234.714,137.630,-50.253,-177.978,5.596,148.375
C06272=1234.709,137.880,-50.274,-177.975,5.597,148.374
C06273=1234.705,138.128,-50.295,-177.973,5.598,148.374
C06274=1234.699,138.378,-50.316,-177.971,5.599,148.373
C06275=1234.695,138.627,-50.336,-177.968,5.601,148.373
C06276=1234.690,138.877,-50.357,-177.965,5.601,148.372
C06277=1234.686,139.126,-50.378,-177.963,5.602,148.372
C06278=1234.681,139.375,-50.399,-177.960,5.604,148.371
C06279=1234.677,139.623,-50.420,-177.958,5.605,148.371
C06280=1234.671,139.872,-50.441,-177.955,5.606,148.370
C06281=1234.667,140.121,-50.461,-177.953,5.607,148.370
C06282=1234.663,140.370,-50.482,-177.950,5.608,148.369
C06283=1234.657,140.620,-50.503,-177.948,5.609,148.369
C06284=1234.653,140.869,-50.523,-177.945,5.611,148.368
C06285=1234.648,141.118,-50.544,-177.942,5.611,148.368
C06286=1234.643,141.367,-50.564,-177.940,5.612,148.367
C06287=1234.638,141.616,-50.585,-177.937,5.614,148.367
C06288=1234.633,141.865,-50.607,-177.935,5.615,148.366
C06289=1234.629,142.114,-50.627,-177.932,5.615,148.366
C06290=1234.624,142.364,-50.649,-177.930,5.617,148.365
C06291=1234.620,142.613,-50.669,-177.927,5.618,148.365
C06292=1234.615,142.862,-50.690,-177.925,5.619,148.364
C06293=1234.610,143.111,-50.710,-177.922,5.620,148.364
C06294=1234.605,143.359,-50.732,-177.920,5.621,148.363
C06295=1234.601,143.608,-50.752,-177.917,5.622,148.363
C06296=1234.596,143.858,-50.773,-177.914,5.624,148.362
C06297=1234.591,144.107,-50.794,-177.912,5.624,148.362
C06298=1234.587,144.356,-50.816,-177.910,5.625,148.361
C06299=1234.582,144.605,-50.837,-177.907,5.627,148.361
C06300=1234.577,144.854,-50.857,-177.904,5.628,148.360
C06301=1234.572,145.103,-50.878,-177.902,5.628,148.360
C06302=1234.567,145.352,-50.900,-177.899,5.630,148.359
C06303=1234.563,145.601,-50.920,-177.897,5.631,148.359
C06304=1234.558,145.851,-50.942,-177.894,5.632,148.358
C06305=1234.554,146.099,-50.963,-177.892,5.634,148.358
C06306=1234.549,146.348,-50.984,-177.889,5.634,148.357
C06307=1234.544,146.598,-51.005,-177.887,5.636,148.357
C06308=1234.540,146.847,-51.025,-177.884,5.637,148.356
C06309=1234.535,147.095,-51.047,-177.882,5.638,148.356
C06310=1234.530,147.345,-51.068,-177.879,5.639,148.355
C06311=1234.526,147.594,-51.089,-177.877,5.640,148.355
C06312=1234.521,147.843,-51.110,-177.874,5.641,148.354
C06313=1234.516,148.092,-51.131,-177.871,5.643,148.354
C06314=1234.511,148.340,-51.152,-177.869,5.644,148.353
C06315=1234.507,148.590,-51.173,-177.866,5.645,148.353
C06316=1234.502,148.839,-51.195,-177.863,5.646,148.352
C06317=1234.497,149.088,-51.216,-177.861,5.647,148.352
C06318=1234.492,149.337,-51.236,-177.858,5.649,148.351
C06319=1234.488,149.586,-51.258,-177.856,5.650,148.351
C06320=1234.483,149.836,-51.279,-177.854,5.650,148.350
C06321=1234.479,150.084,-51.300,-177.851,5.652,148.350
C06322=1234.474,150.333,-51.321,-177.849,5.653,148.349
C06323=1234.469,150.582,-51.343,-177.846,5.654,148.349
C06324=1234.464,150.832,-51.364,-177.843,5.655,148.348
C06325=1234.460,151.080,-51.386,-177.841,5.656,148.348
C06326=1234.455,151.330,-51.407,-177.838,5.658,148.347
C06327=1234.450,151.578,-51.428,-177.836,5.659,148.347
C06328=1234.445,151.828,-51.450,-177.833,5.660,148.346
C06329=1234.441,152.077,-51.471,-177.830,5.661,148.346
C06330=1234.436,152.326,-51.492,-177.828,5.662,148.345
C06331=1234.431,152.574,-51.513,-177.825,5.664,148.345
C06332=1234.427,152.824,-51.535,-177.823,5.665,148.344
C06333=1234.422,153.073,-51.556,-177.820,5.666,148.344
C06334=1234.417,153.322,-51.578,-177.818,5.667,148.343
C06335=1234.412,153.571,-51.599,-177.816,5.668,148.343
C06336=1234.408,153.820,-51.620,-177.813,5.670,148.342
C06337=1234.403,154.069,-51.641,-177.810,5.671,148.342
C06338=1234.398,154.318,-51.663,-177.807,5.672,148.341
C06339=1234.394,154.567,-51.685,-177.805,5.673,148.341
C06340=1234.389,154.816,-51.706,-177.803,5.674,148.340
C06341=1234.384,155.065,-51.728,-177.800,5.676,148.340
C06342=1234.380,155.314,-51.750,-177.798,5.677,148.340
C06343=1234.375,155.563,-51.770,-177.795,5.678,148.339
C06344=1234.370,155.812,-51.792,-177.793,5.679,148.339
C06345=1234.366,156.061,-51.814,-177.789,5.681,148.338
C06346=1234.361,156.311,-51.835,-177.787,5.682,148.338
C06347=1234.356,156.559,-51.857,-177.785,5.682,148.337
C06348=1234.352,156.809,-51.879,-177.782,5.684,148.337
C06349=1234.347,157.057,-51.900,-177.780,5.685,148.336
C06350=1234.342,157.307,-51.921,-177.777,5.687,148.336
C06351=1234.337,157.556,-51.943,-177.775,5.688,148.335
C06352=1234.333,157.805,-51.965,-177.772,5.689,148.335
C06353=1234.328,158.053,-51.987,-177.769,5.690,148.334
C06354=1234.323,158.303,-52.008,-177.767,5.691,148.334
C06355=1234.318,158.552,-52.030,-177.764,5.693,148.333
C06356=1234.314,158.800,-52.051,-177.762,5.694,148.333
C06357=1234.310,159.049,-52.073,-177.759,5.695,148.332
C06358=1234.305,159.298,-52.094,-177.757,5.696,148.332
C06359=1234.300,159.567,-52.118,-177.754,5.698,148.331
C06360=1234.294,159.837,-52.141,-177.751,5.699,148.331
C06361=1234.290,160.105,-52.165,-177.748,5.700,148.330
C06362=1234.285,160.375,-52.188,-177.746,5.702,148.330
C06363=1234.280,160.624,-52.210,-177.743,5.703,148.329
C06364=1234.275,160.873,-52.232,-177.741,5.704,148.329
C06365=1234.271,161.122,-52.254,-177.738,5.705,148.328
C06366=1234.266,161.371,-52.275,-177.735,5.707,148.328
C06367=1234.261,161.621,-52.297,-177.733,5.708,148.328
C06368=1234.256,161.869,-52.319,-177.730,5.709,148.327
C06369=1234.252,162.118,-52.340,-177.728,5.710,148.327
C06370=1234.247,162.367,-52.362,-177.725,5.711,148.326
C06371=1234.242,162.616,-52.384,-177.723,5.713,148.326
C06372=1234.237,162.865,-52.407,-177.721,5.714,148.325
C06373=1234.233,163.114,-52.428,-177.718,5.715,148.325
C06374=1234.228,163.363,-52.450,-177.715,5.716,148.324
C06375=1234.223,163.612,-52.472,-177.712,5.718,148.324
C06376=1234.219,163.861,-52.494,-177.710,5.719,148.323
C06377=1234.214,164.110,-52.516,-177.708,5.721,148.323
C06378=1234.209,164.359,-52.537,-177.705,5.721,148.322
C06379=1234.205,164.608,-52.559,-177.702,5.723,148.322
C06380=1234.200,164.857,-52.581,-177.700,5.724,148.322
C06381=1234.196,165.106,-52.603,-177.697,5.726,148.321
C06382=1234.190,165.355,-52.625,-177.695,5.727,148.321
C06383=1234.186,165.604,-52.647,-177.692,5.728,148.320
C06384=1234.181,165.853,-52.669,-177.690,5.729,148.320
C06385=1234.177,166.102,-52.691,-177.687,5.731,148.319
C06386=1234.172,166.350,-52.714,-177.684,5.732,148.319
C06387=1234.168,166.600,-52.736,-177.682,5.734,148.318
C06388=1234.163,166.849,-52.758,-177.680,5.735,148.318
C06389=1234.158,167.098,-52.780,-177.677,5.736,148.317
C06390=1234.153,167.347,-52.802,-177.674,5.737,148.317
C06391=1234.149,167.596,-52.824,-177.672,5.738,148.316
C06392=1234.144,167.845,-52.845,-177.669,5.740,148.316
C06393=1234.139,168.094,-52.868,-177.667,5.741,148.316
C06394=1234.135,168.343,-52.891,-177.664,5.742,148.315
C06395=1234.130,168.592,-52.913,-177.662,5.743,148.315
C06396=1234.126,168.841,-52.935,-177.659,5.745,148.314
C06397=1234.121,169.090,-52.956,-177.657,5.746,148.314
C06398=1234.116,169.339,-52.979,-177.654,5.748,148.313
C06399=1234.112,169.587,-53.001,-177.651,5.749,148.313
C06400=1234.107,169.837,-53.023,-177.649,5.750,148.312
C06401=1234.102,170.086,-53.046,-177.646,5.752,148.312
C06402=1234.098,170.335,-53.068,-177.644,5.753,148.311
C06403=1234.093,170.583,-53.090,-177.641,5.754,148.311
C06404=1234.089,170.832,-53.112,-177.639,5.755,148.311
C06405=1234.084,171.082,-53.135,-177.636,5.757,148.310
C06406=1234.079,171.331,-53.156,-177.634,5.758,148.310
C06407=1234.075,171.579,-53.179,-177.631,5.760,148.309
C06408=1234.069,171.828,-53.201,-177.629,5.761,148.309
C06409=1234.065,172.078,-53.224,-177.626,5.762,148.308
C06410=1234.061,172.326,-53.246,-177.624,5.763,148.308
C06411=1234.055,172.575,-53.269,-177.621,5.765,148.307
C06412=1234.051,172.825,-53.291,-177.618,5.766,148.307
C06413=1234.047,173.073,-53.313,-177.616,5.768,148.307
C06414=1234.042,173.322,-53.336,-177.614,5.769,148.306
C06415=1234.037,173.572,-53.358,-177.610,5.770,148.306
C06416=1234.033,173.820,-53.380,-177.608,5.771,148.305
C06417=1234.028,174.069,-53.403,-177.606,5.773,148.305
C06418=1234.023,174.317,-53.425,-177.603,5.774,148.304
C06419=1234.019,174.567,-53.447,-177.601,5.776,148.304
C06420=1234.014,174.816,-53.470,-177.598,5.777,148.303
C06421=1234.009,175.064,-53.492,-177.595,5.778,148.303
C06422=1234.004,175.314,-53.515,-177.593,5.780,148.303
C06423=1234.000,175.563,-53.538,-177.591,5.781,148.302
C06424=1233.995,175.812,-53.560,-177.587,5.782,148.302
C06425=1233.991,176.060,-53.583,-177.585,5.783,148.301
C06426=1233.987,176.310,-53.605,-177.583,5.785,148.301
C06427=1233.981,176.558,-53.628,-177.580,5.786,148.300
C06428=1233.977,176.807,-53.650,-177.577,5.788,148.300
C06429=1233.972,177.056,-53.673,-177.575,5.789,148.299
C06430=1233.967,177.305,-53.695,-177.573,5.791,148.299
C06431=1233.963,177.554,-53.718,-177.570,5.792,148.299
C06432=1233.958,177.803,-53.740,-177.567,5.793,148.298
C06433=1233.953,178.052,-53.763,-177.565,5.795,148.298
C06434=1233.949,178.301,-53.785,-177.562,5.796,148.297
C06435=1233.944,178.550,-53.809,-177.560,5.798,148.297
C06436=1233.940,178.799,-53.831,-177.558,5.799,148.296
C06437=1233.935,179.048,-53.854,-177.554,5.800,148.296
C06438=1233.931,179.296,-53.876,-177.552,5.801,148.295
C06439=1233.926,179.546,-53.899,-177.550,5.803,148.295
C06440=1233.921,179.794,-53.921,-177.547,5.805,148.295
C06441=1233.916,180.043,-53.945,-177.544,5.805,148.294
C06442=1233.912,180.293,-53.967,-177.542,5.807,148.294
C06443=1233.907,180.542,-53.990,-177.540,5.808,148.293
C06444=1233.903,180.790,-54.013,-177.537,5.810,148.293
C06445=1233.898,181.039,-54.035,-177.534,5.811,148.292
C06446=1233.894,181.288,-54.058,-177.532,5.813,148.292
C06447=1233.889,181.537,-54.081,-177.529,5.815,148.292
C06448=1233.884,181.786,-54.104,-177.527,5.815,148.291
C06449=1233.880,182.035,-54.126,-177.524,5.817,148.291
C06450=1233.875,182.284,-54.150,-177.522,5.818,148.290
C06451=1233.871,182.532,-54.173,-177.519,5.820,148.290
C06452=1233.865,182.781,-54.195,-177.516,5.821,148.289
C06453=1233.861,183.030,-54.218,-177.514,5.823,148.289
C06454=1233.857,183.279,-54.241,-177.511,5.824,148.289
C06455=1233.852,183.528,-54.264,-177.509,5.825,148.288
C06456=1233.848,183.777,-54.286,-177.506,5.827,148.288
C06457=1233.842,184.026,-54.309,-177.503,5.829,148.287
C06458=1233.838,184.275,-54.333,-177.501,5.830,148.287
C06459=1233.834,184.524,-54.355,-177.498,5.831,148.286
C06460=1233.829,184.773,-54.379,-177.496,5.832,148.286
C06461=1233.824,185.022,-54.401,-177.494,5.834,148.286
C06462=1233.819,185.270,-54.424,-177.491,5.836,148.285
C06463=1233.814,185.540,-54.449,-177.488,5.837,148.285
C06464=1233.809,185.810,-54.474,-177.486,5.839,148.284
C06465=1233.805,186.079,-54.499,-177.483,5.840,148.284
C06466=1233.800,186.349,-54.524,-177.480,5.842,148.284
C06467=1233.795,186.598,-54.548,-177.478,5.843,148.283
C06468=1233.790,186.847,-54.570,-177.475,5.844,148.283
C06469=1233.786,187.096,-54.593,-177.472,5.846,148.282
C06470=1233.781,187.345,-54.616,-177.470,5.847,148.282
C06471=1233.776,187.594,-54.640,-177.467,5.849,148.281
C06472=1233.772,187.843,-54.662,-177.464,5.851,148.281
C06473=1233.768,188.092,-54.686,-177.462,5.852,148.281
C06474=1233.763,188.341,-54.709,-177.459,5.854,148.280
C06475=1233.758,188.589,-54.732,-177.457,5.855,148.280
C06476=1233.753,188.838,-54.755,-177.454,5.856,148.279
C06477=1233.749,189.087,-54.778,-177.452,5.858,148.279
C06478=1233.744,189.336,-54.802,-177.450,5.859,148.279
C06479=1233.739,189.585,-54.825,-177.447,5.861,148.278
C06480=1233.735,189.834,-54.848,-177.444,5.863,148.278
C06481=1233.731,190.083,-54.871,-177.442,5.863,148.277
C06482=1233.726,190.332,-54.894,-177.439,5.865,148.277
C06483=1233.721,190.581,-54.918,-177.437,5.866,148.276
C06484=1233.716,190.829,-54.941,-177.434,5.868,148.276
C06485=1233.711,191.078,-54.964,-177.431,5.870,148.276
C06486=1233.707,191.326,-54.988,-177.429,5.871,148.275
C06487=1233.702,191.575,-55.012,-177.426,5.872,148.275
C06488=1233.698,191.824,-55.034,-177.424,5.874,148.275
C06489=1233.694,192.073,-55.058,-177.422,5.875,148.274
C06490=1233.689,192.322,-55.081,-177.419,5.877,148.274
C06491=1233.684,192.571,-55.104,-177.416,5.879,148.273
C06492=1233.680,192.820,-55.128,-177.414,5.880,148.273
C06493=1233.675,193.069,-55.151,-177.411,5.882,148.272
C06494=1233.670,193.318,-55.175,-177.409,5.883,148.272
C06495=1233.666,193.567,-55.199,-177.406,5.884,148.272
C06496=1233.662,193.815,-55.221,-177.403,5.886,148.271
C06497=1233.657,194.065,-55.245,-177.401,5.888,148.271
C06498=1233.652,194.314,-55.268,-177.399,5.889,148.270
C06499=1233.648,194.562,-55.292,-177.396,5.891,148.270
C06500=1233.643,194.811,-55.315,-177.393,5.892,148.270
C06501=1233.638,195.059,-55.338,-177.391,5.893,148.269
C06502=1233.633,195.308,-55.362,-177.388,5.895,148.269
C06503=1233.629,195.557,-55.386,-177.386,5.897,148.269
C06504=1233.624,195.806,-55.409,-177.383,5.898,148.268
C06505=1233.620,196.055,-55.433,-177.380,5.900,148.268
C06506=1233.615,196.304,-55.456,-177.378,5.901,148.267
C06507=1233.610,196.552,-55.480,-177.376,5.902,148.267
C06508=1233.606,196.801,-55.503,-177.373,5.904,148.266
C06509=1233.602,197.051,-55.527,-177.370,5.906,148.266
C06510=1233.597,197.299,-55.551,-177.368,5.907,148.266
C06511=1233.593,197.548,-55.575,-177.365,5.909,148.265
C06512=1233.588,197.798,-55.598,-177.362,5.911,148.265
C06513=1233.583,198.046,-55.622,-177.360,5.912,148.264
C06514=1233.579,198.295,-55.645,-177.358,5.913,148.264
C06515=1233.574,198.543,-55.669,-177.355,5.915,148.264
C06516=1233.570,198.792,-55.693,-177.353,5.916,148.263
C06517=1233.565,199.041,-55.716,-177.350,5.918,148.263
C06518=1233.561,199.290,-55.740,-177.347,5.920,148.263
C06519=1233.556,199.539,-55.764,-177.345,5.922,148.262
C06520=1233.551,199.787,-55.788,-177.343,5.923,148.262
C06521=1233.547,200.036,-55.811,-177.340,5.924,148.261
C06522=1233.542,200.285,-55.836,-177.337,5.926,148.261
C06523=1233.537,200.534,-55.859,-177.335,5.927,148.261
C06524=1233.533,200.782,-55.883,-177.332,5.929,148.260
C06525=1233.528,201.032,-55.906,-177.329,5.931,148.260
C06526=1233.523,201.280,-55.931,-177.327,5.932,148.259
C06527=1233.519,201.530,-55.954,-177.325,5.934,148.259
C06528=1233.515,201.778,-55.978,-177.322,5.935,148.259
C06529=1233.510,202.027,-56.002,-177.319,5.937,148.258
C06530=1233.505,202.276,-56.026,-177.317,5.938,148.258
C06531=1233.500,202.525,-56.050,-177.314,5.940,148.258
C06532=1233.496,202.773,-56.074,-177.312,5.942,148.257
C06533=1233.491,203.022,-56.097,-177.310,5.943,148.257
C06534=1233.487,203.271,-56.121,-177.306,5.944,148.256
C06535=1233.482,203.520,-56.145,-177.304,5.946,148.256
C06536=1233.478,203.769,-56.170,-177.301,5.948,148.256
C06537=1233.473,204.018,-56.194,-177.299,5.949,148.255
C06538=1233.469,204.267,-56.217,-177.296,5.951,148.255
C06539=1233.464,204.515,-56.241,-177.294,5.953,148.255
C06540=1233.460,204.763,-56.265,-177.291,5.955,148.254
C06541=1233.454,205.013,-56.289,-177.289,5.955,148.254
C06542=1233.450,205.261,-56.313,-177.286,5.957,148.253
C06543=1233.446,205.510,-56.338,-177.283,5.959,148.253
C06544=1233.441,205.759,-56.361,-177.281,5.961,148.253
C06545=1233.437,206.008,-56.385,-177.279,5.962,148.252
C06546=1233.432,206.256,-56.410,-177.276,5.964,148.252
C06547=1233.427,206.506,-56.433,-177.273,5.966,148.252
C06548=1233.423,206.755,-56.458,-177.271,5.967,148.251
C06549=1233.418,207.003,-56.482,-177.268,5.968,148.251
C06550=1233.414,207.252,-56.506,-177.266,5.970,148.250
C06551=1233.409,207.501,-56.530,-177.263,5.972,148.250
C06552=1233.405,207.749,-56.554,-177.261,5.973,148.250
C06553=1233.400,207.998,-56.578,-177.258,5.975,148.249
C06554=1233.396,208.247,-56.603,-177.256,5.977,148.249
C06555=1233.392,208.495,-56.627,-177.253,5.979,148.249
C06556=1233.386,208.745,-56.651,-177.251,5.980,148.248
C06557=1233.382,208.993,-56.675,-177.248,5.982,148.248
C06558=1233.378,209.242,-56.699,-177.245,5.983,148.247
C06559=1233.373,209.491,-56.724,-177.243,5.985,148.247
C06560=1233.368,209.739,-56.748,-177.240,5.987,148.247
C06561=1233.364,209.988,-56.772,-177.238,5.988,148.246
C06562=1233.359,210.238,-56.797,-177.235,5.990,148.246
C06563=1233.355,210.486,-56.821,-177.233,5.992,148.246
C06564=1233.350,210.735,-56.845,-177.230,5.993,148.245
C06565=1233.345,210.983,-56.869,-177.228,5.994,148.245
C06566=1233.341,211.233,-56.894,-177.225,5.996,148.245
C06567=1233.336,211.503,-56.921,-177.222,5.998,148.244
C06568=1233.331,211.774,-56.947,-177.220,6.000,148.244
C06569=1233.326,212.044,-56.973,-177.217,6.002,148.243
C06570=1233.321,212.314,-57.000,-177.214,6.003,148.243
C06571=1233.317,212.563,-57.024,-177.211,6.005,148.242
C06572=1233.312,212.811,-57.048,-177.209,6.007,148.242
C06573=1233.307,213.060,-57.073,-177.206,6.009,148.242
C06574=1233.303,213.309,-57.098,-177.204,6.010,148.241
C06575=1233.298,213.558,-57.122,-177.201,6.012,148.241
C06576=1233.294,213.806,-57.146,-177.199,6.013,148.241
C06577=1233.289,214.056,-57.171,-177.196,6.015,148.240
C06578=1233.285,214.304,-57.195,-177.193,6.017,148.240
C06579=1233.280,214.553,-57.220,-177.191,6.018,148.240
C06580=1233.275,214.801,-57.244,-177.189,6.020,148.239
C06581=1233.271,215.051,-57.269,-177.186,6.022,148.239
C06582=1233.267,215.299,-57.293,-177.183,6.024,148.239
C06583=1233.261,215.548,-57.318,-177.180,6.025,148.238
C06584=1233.258,215.796,-57.343,-177.178,6.026,148.238
C06585=1233.253,216.045,-57.368,-177.176,6.028,148.238
C06586=1233.249,216.294,-57.392,-177.173,6.030,148.237
C06587=1233.244,216.543,-57.417,-177.170,6.032,148.237
C06588=1233.239,216.791,-57.441,-177.168,6.034,148.237
C06589=1233.235,217.041,-57.466,-177.166,6.035,148.236
C06590=1233.230,217.290,-57.491,-177.163,6.037,148.236
C06591=1233.226,217.537,-57.515,-177.160,6.039,148.236
C06592=1233.221,217.787,-57.540,-177.158,6.041,148.235
C06593=1233.217,218.035,-57.565,-177.155,6.042,148.235
C06594=1233.212,218.284,-57.589,-177.153,6.043,148.234
C06595=1233.207,218.533,-57.614,-177.150,6.045,148.234
C06596=1233.203,218.781,-57.639,-177.148,6.047,148.234
C06597=1233.198,219.031,-57.664,-177.145,6.049,148.233
C06598=1233.194,219.279,-57.688,-177.142,6.051,148.233
C06599=1233.189,219.528,-57.713,-177.139,6.053,148.233
C06600=1233.185,219.776,-57.739,-177.137,6.054,148.232
C06601=1233.180,220.025,-57.763,-177.135,6.055,148.232
C06602=1233.176,220.274,-57.788,-177.132,6.057,148.232
C06603=1233.171,220.522,-57.813,-177.129,6.059,148.231
C06604=1233.167,220.772,-57.838,-177.127,6.061,148.231
C06605=1233.162,221.020,-57.862,-177.124,6.063,148.231
C06606=1233.157,221.268,-57.888,-177.122,6.064,148.230
C06607=1233.153,221.517,-57.912,-177.120,6.066,148.230
C06608=1233.148,221.766,-57.937,-177.117,6.068,148.230
C06609=1233.144,222.015,-57.962,-177.114,6.070,148.229
C06610=1233.140,222.263,-57.987,-177.112,6.071,148.229
C06611=1233.135,222.512,-58.012,-177.110,6.072,148.229
C06612=1233.130,222.761,-58.037,-177.107,6.074,148.228
C06613=1233.126,223.010,-58.062,-177.104,6.076,148.228
C06614=1233.122,223.258,-58.087,-177.102,6.078,148.228
C06615=1233.117,223.508,-58.112,-177.099,6.080,148.227
C06616=1233.112,223.756,-58.137,-177.096,6.082,148.227
C06617=1233.108,224.005,-58.162,-177.094,6.083,148.227
C06618=1233.104,224.253,-58.187,-177.092,6.085,148.226
C06619=1233.099,224.502,-58.212,-177.089,6.087,148.226
C06620=1233.094,224.750,-58.237,-177.087,6.088,148.226
C06621=1233.090,225.000,-58.262,-177.084,6.090,148.225
C06622=1233.086,225.248,-58.287,-177.081,6.092,148.225
C06623=1233.081,225.497,-58.312,-177.079,6.094,148.225
C06624=1233.076,225.745,-58.338,-177.077,6.095,148.224
C06625=1233.072,225.995,-58.363,-177.074,6.097,148.224
C06626=1233.067,226.243,-58.388,-177.071,6.099,148.224
C06627=1233.063,226.492,-58.413,-177.069,6.101,148.223
C06628=1233.058,226.740,-58.438,-177.066,6.103,148.223
C06629=1233.054,226.989,-58.463,-177.064,6.105,148.223
C06630=1233.049,227.237,-58.488,-177.061,6.106,148.222
C06631=1233.045,227.486,-58.514,-177.059,6.107,148.222
C06632=1233.040,227.735,-58.539,-177.056,6.109,148.222
C06633=1233.035,227.984,-58.564,-177.054,6.111,148.221
C06634=1233.031,228.232,-58.590,-177.051,6.113,148.221
C06635=1233.027,228.481,-58.614,-177.048,6.115,148.221
C06636=1233.023,228.730,-58.640,-177.046,6.117,148.220
C06637=1233.018,228.978,-58.665,-177.044,6.118,148.220
C06638=1233.013,229.227,-58.690,-177.041,6.120,148.220
C06639=1233.008,229.475,-58.716,-177.038,6.122,148.219
C06640=1233.004,229.724,-58.742,-177.036,6.123,148.219
C06641=1232.999,229.973,-58.766,-177.033,6.125,148.219
C06642=1232.995,230.222,-58.792,-177.031,6.128,148.219
C06643=1232.991,230.471,-58.818,-177.028,6.129,148.218
C06644=1232.986,230.719,-58.843,-177.026,6.130,148.218
C06645=1232.981,230.968,-58.868,-177.024,6.132,148.218
C06646=1232.976,231.216,-58.894,-177.021,6.134,148.217
C06647=1232.972,231.465,-58.919,-177.019,6.136,148.217
C06648=1232.968,231.714,-58.945,-177.016,6.138,148.217
C06649=1232.963,231.963,-58.970,-177.013,6.140,148.216
C06650=1232.959,232.211,-58.996,-177.011,6.142,148.216
C06651=1232.954,232.460,-59.021,-177.008,6.144,148.216
C06652=1232.950,232.708,-59.047,-177.006,6.145,148.215
C06653=1232.945,232.957,-59.072,-177.003,6.147,148.215
C06654=1232.941,233.206,-59.098,-177.001,6.148,148.215
C06655=1232.936,233.455,-59.123,-176.998,6.150,148.214
C06656=1232.932,233.703,-59.149,-176.996,6.152,148.214
C06657=1232.927,233.951,-59.174,-176.993,6.154,148.214
C06658=1232.923,234.200,-59.200,-176.991,6.156,148.214
C06659=1232.919,234.449,-59.225,-176.988,6.158,148.213
C06660=1232.914,234.697,-59.251,-176.986,6.160,148.213
C06661=1232.909,234.946,-59.277,-176.983,6.161,148.213
C06662=1232.905,235.195,-59.302,-176.981,6.163,148.212
C06663=1232.901,235.444,-59.328,-176.978,6.165,148.212
C06664=1232.896,235.692,-59.353,-176.976,6.167,148.212
C06665=1232.892,235.941,-59.379,-176.973,6.169,148.211
C06666=1232.888,236.189,-59.405,-176.970,6.170,148.211
C06667=1232.883,236.437,-59.430,-176.968,6.172,148.211
C06668=1232.878,236.687,-59.457,-176.965,6.174,148.210
C06669=1232.874,236.935,-59.482,-176.963,6.176,148.210
C06670=1232.869,237.183,-59.508,-176.961,6.177,148.210
C06671=1232.864,237.455,-59.536,-176.957,6.180,148.210
C06672=1232.860,237.727,-59.564,-176.955,6.182,148.209
C06673=1232.855,237.998,-59.592,-176.952,6.184,148.209
C06674=1232.850,238.270,-59.620,-176.949,6.186,148.209
C06675=1232.845,238.518,-59.646,-176.947,6.187,148.208
C06676=1232.841,238.767,-59.672,-176.945,6.190,148.208
C06677=1232.836,239.016,-59.698,-176.942,6.191,148.208
C06678=1232.832,239.265,-59.724,-176.940,6.193,148.208
C06679=1232.827,239.512,-59.750,-176.937,6.195,148.207
C06680=1232.823,239.761,-59.775,-176.934,6.197,148.207
C06681=1232.819,240.010,-59.801,-176.932,6.198,148.207
C06682=1232.814,240.259,-59.828,-176.930,6.200,148.206
C06683=1232.809,240.508,-59.853,-176.927,6.202,148.206
C06684=1232.805,240.756,-59.879,-176.924,6.204,148.206
C06685=1232.800,241.004,-59.904,-176.922,6.206,148.206
C06686=1232.796,241.253,-59.932,-176.920,6.208,148.205
C06687=1232.792,241.502,-59.957,-176.917,6.210,148.205
C06688=1232.787,241.750,-59.983,-176.914,6.212,148.205
C06689=1232.782,241.999,-60.008,-176.912,6.214,148.204
C06690=1232.778,242.247,-60.035,-176.909,6.215,148.204
C06691=1232.774,242.496,-60.061,-176.907,6.217,148.204
C06692=1232.769,242.745,-60.087,-176.904,6.220,148.204
C06693=1232.764,242.993,-60.113,-176.902,6.221,148.203
C06694=1232.760,243.241,-60.139,-176.900,6.222,148.203
C06695=1232.756,243.490,-60.165,-176.897,6.224,148.203
C06696=1232.751,243.739,-60.191,-176.895,6.226,148.202
C06697=1232.747,243.987,-60.218,-176.892,6.228,148.202
C06698=1232.743,244.236,-60.244,-176.890,6.230,148.202
C06699=1232.737,244.485,-60.270,-176.887,6.232,148.202
C06700=1232.733,244.733,-60.296,-176.885,6.234,148.201
C06701=1232.729,244.982,-60.322,-176.882,6.236,148.201
C06702=1232.724,245.231,-60.348,-176.879,6.238,148.201
C06703=1232.720,245.479,-60.375,-176.877,6.240,148.200
C06704=1232.716,245.728,-60.400,-176.874,6.242,148.200
C06705=1232.711,245.976,-60.428,-176.872,6.244,148.200
C06706=1232.706,246.224,-60.453,-176.869,6.246,148.200
C06707=1232.701,246.474,-60.479,-176.867,6.248,148.199
C06708=1232.697,246.722,-60.506,-176.864,6.250,148.199
C06709=1232.693,246.971,-60.531,-176.862,6.251,148.199
C06710=1232.688,247.219,-60.559,-176.860,6.253,148.199
C06711=1232.684,247.468,-60.584,-176.857,6.255,148.198
C06712=1232.680,247.716,-60.611,-176.855,6.257,148.198
C06713=1232.675,247.965,-60.637,-176.852,6.258,148.198
C06714=1232.671,248.214,-60.664,-176.850,6.260,148.197
C06715=1232.667,248.462,-60.690,-176.847,6.263,148.197
C06716=1232.662,248.710,-60.716,-176.845,6.264,148.197
C06717=1232.657,248.959,-60.742,-176.842,6.266,148.197
C06718=1232.653,249.207,-60.769,-176.840,6.268,148.196
C06719=1232.648,249.456,-60.795,-176.837,6.270,148.196
C06720=1232.644,249.704,-60.822,-176.835,6.272,148.196
C06721=1232.640,249.953,-60.849,-176.832,6.274,148.196
C06722=1232.635,250.202,-60.874,-176.830,6.276,148.195
C06723=1232.631,250.450,-60.902,-176.827,6.278,148.195
C06724=1232.626,250.699,-60.927,-176.824,6.280,148.195
C06725=1232.622,250.948,-60.954,-176.822,6.282,148.195
C06726=1232.617,251.196,-60.981,-176.820,6.284,148.194
C06727=1232.613,251.445,-61.007,-176.817,6.286,148.194
C06728=1232.608,251.693,-61.034,-176.815,6.288,148.194
C06729=1232.604,251.942,-61.061,-176.812,6.290,148.193
C06730=1232.599,252.191,-61.087,-176.810,6.292,148.193
C06731=1232.595,252.439,-61.113,-176.807,6.294,148.193
C06732=1232.591,252.687,-61.141,-176.805,6.296,148.193
C06733=1232.586,252.936,-61.167,-176.802,6.297,148.192
C06734=1232.582,253.185,-61.193,-176.800,6.300,148.192
C06735=1232.577,253.433,-61.220,-176.797,6.302,148.192
C06736=1232.573,253.681,-61.247,-176.795,6.303,148.192
C06737=1232.568,253.930,-61.273,-176.792,6.305,148.191
C06738=1232.564,254.179,-61.300,-176.790,6.308,148.191
C06739=1232.560,254.427,-61.327,-176.787,6.309,148.191
C06740=1232.555,254.676,-61.354,-176.785,6.311,148.191
C06741=1232.551,254.924,-61.380,-176.782,6.313,148.190
C06742=1232.546,255.173,-61.407,-176.780,6.315,148.190
C06743=1232.542,255.421,-61.434,-176.777,6.317,148.190
C06744=1232.538,255.670,-61.460,-176.775,6.319,148.190
C06745=1232.533,255.918,-61.487,-176.772,6.321,148.189
C06746=1232.528,256.167,-61.514,-176.770,6.323,148.189
C06747=1232.524,256.415,-61.540,-176.767,6.325,148.189
C06748=1232.520,256.664,-61.567,-176.765,6.327,148.189
C06749=1232.515,256.912,-61.594,-176.762,6.329,148.188
C06750=1232.510,257.161,-61.621,-176.760,6.331,148.188
C06751=1232.506,257.409,-61.648,-176.758,6.333,148.188
C06752=1232.502,257.658,-61.675,-176.755,6.335,148.188
C06753=1232.498,257.907,-61.702,-176.753,6.337,148.188
C06754=1232.493,258.155,-61.729,-176.750,6.339,148.187
C06755=1232.489,258.403,-61.756,-176.748,6.341,148.187
C06756=1232.484,258.652,-61.783,-176.745,6.343,148.187
C06757=1232.480,258.900,-61.810,-176.743,6.345,148.187
C06758=1232.475,259.149,-61.837,-176.740,6.347,148.186
C06759=1232.471,259.397,-61.863,-176.738,6.349,148.186
C06760=1232.466,259.646,-61.890,-176.736,6.351,148.186
C06761=1232.462,259.894,-61.917,-176.733,6.353,148.186
C06762=1232.457,260.143,-61.945,-176.730,6.355,148.185
C06763=1232.453,260.392,-61.972,-176.728,6.357,148.185
C06764=1232.449,260.640,-61.998,-176.726,6.359,148.185
C06765=1232.444,260.888,-62.025,-176.723,6.361,148.185
C06766=1232.440,261.137,-62.053,-176.720,6.363,148.184
C06767=1232.435,261.385,-62.080,-176.718,6.365,148.184
C06768=1232.431,261.634,-62.107,-176.716,6.367,148.184
C06769=1232.426,261.882,-62.134,-176.713,6.369,148.184
C06770=1232.423,262.131,-62.161,-176.711,6.371,148.184
C06771=1232.418,262.380,-62.188,-176.708,6.373,148.183
C06772=1232.414,262.628,-62.215,-176.706,6.375,148.183
C06773=1232.409,262.876,-62.242,-176.704,6.377,148.183
C06774=1232.404,263.125,-62.270,-176.701,6.379,148.183
C06775=1232.400,263.397,-62.299,-176.698,6.382,148.182
C06776=1232.394,263.670,-62.330,-176.695,6.384,148.182
C06777=1232.390,263.943,-62.359,-176.693,6.385,148.182
C06778=1232.386,264.216,-62.389,-176.690,6.388,148.182
C06779=1232.381,264.464,-62.416,-176.687,6.390,148.181
C06780=1232.377,264.712,-62.443,-176.685,6.392,148.181
C06781=1232.372,264.960,-62.471,-176.683,6.394,148.181
C06782=1232.367,265.209,-62.498,-176.680,6.396,148.181
C06783=1232.363,265.458,-62.525,-176.678,6.398,148.180
C06784=1232.359,265.706,-62.553,-176.675,6.400,148.180
C06785=1232.354,265.955,-62.580,-176.673,6.402,148.180
C06786=1232.350,266.203,-62.607,-176.671,6.405,148.180
C06787=1232.345,266.451,-62.635,-176.668,6.406,148.180
C06788=1232.341,266.700,-62.662,-176.665,6.408,148.179
C06789=1232.337,266.949,-62.689,-176.663,6.411,148.179
C06790=1232.332,267.197,-62.716,-176.661,6.412,148.179
C06791=1232.328,267.445,-62.744,-176.658,6.414,148.179
C06792=1232.324,267.694,-62.771,-176.656,6.417,148.179
C06793=1232.319,267.942,-62.799,-176.653,6.419,148.178
C06794=1232.315,268.191,-62.826,-176.651,6.422,148.178
C06795=1232.310,268.439,-62.853,-176.648,6.423,148.178
C06796=1232.306,268.688,-62.882,-176.646,6.425,148.178
C06797=1232.301,268.936,-62.909,-176.643,6.428,148.178
C06798=1232.297,269.184,-62.936,-176.641,6.429,148.177
C06799=1232.292,269.432,-62.963,-176.639,6.432,148.177
C06800=1232.288,269.681,-62.992,-176.636,6.434,148.177
C06801=1232.283,269.930,-63.019,-176.634,6.435,148.177
C06802=1232.279,270.178,-63.046,-176.631,6.438,148.177
C06803=1232.275,270.427,-63.074,-176.629,6.440,148.176
C06804=1232.270,270.675,-63.101,-176.627,6.442,148.176
C06805=1232.266,270.923,-63.129,-176.624,6.445,148.176
C06806=1232.262,271.172,-63.157,-176.621,6.446,148.176
C06807=1232.257,271.420,-63.184,-176.619,6.449,148.176
C06808=1232.253,271.668,-63.212,-176.616,6.451,148.175
C06809=1232.248,271.918,-63.240,-176.614,6.453,148.175
C06810=1232.244,272.166,-63.268,-176.612,6.455,148.175
C06811=1232.239,272.414,-63.295,-176.609,6.457,148.175
C06812=1232.236,272.663,-63.323,-176.607,6.459,148.175
C06813=1232.231,272.911,-63.350,-176.604,6.461,148.174
C06814=1232.227,273.159,-63.378,-176.602,6.463,148.174
C06815=1232.222,273.408,-63.407,-176.600,6.465,148.174
C06816=1232.217,273.656,-63.434,-176.597,6.468,148.174
C06817=1232.213,273.904,-63.462,-176.594,6.470,148.174
C06818=1232.209,274.153,-63.490,-176.592,6.472,148.174
C06819=1232.205,274.401,-63.517,-176.590,6.474,148.173
C06820=1232.200,274.650,-63.545,-176.587,6.476,148.173
C06821=1232.196,274.898,-63.573,-176.585,6.478,148.173
C06822=1232.191,275.147,-63.600,-176.582,6.480,148.173
C06823=1232.187,275.395,-63.629,-176.580,6.482,148.173
C06824=1232.182,275.643,-63.657,-176.578,6.484,148.172
C06825=1232.178,275.892,-63.684,-176.575,6.487,148.172
C06826=1232.174,276.140,-63.712,-176.572,6.489,148.172
C06827=1232.170,276.388,-63.740,-176.570,6.491,148.172
C06828=1232.165,276.637,-63.769,-176.568,6.493,148.172
C06829=1232.160,276.886,-63.796,-176.566,6.495,148.172
C06830=1232.156,277.134,-63.823,-176.563,6.497,148.171
C06831=1232.152,277.383,-63.852,-176.561,6.499,148.171
C06832=1232.147,277.630,-63.880,-176.558,6.501,148.171
C06833=1232.143,277.879,-63.908,-176.556,6.504,148.171
C06834=1232.139,278.127,-63.936,-176.553,6.506,148.171
C06835=1232.134,278.376,-63.964,-176.551,6.508,148.171
C06836=1232.130,278.624,-63.992,-176.548,6.510,148.170
C06837=1232.126,278.873,-64.020,-176.546,6.513,148.170
C06838=1232.121,279.121,-64.048,-176.544,6.514,148.170
C06839=1232.117,279.369,-64.076,-176.541,6.517,148.170
C06840=1232.112,279.618,-64.105,-176.539,6.519,148.170
C06841=1232.108,279.866,-64.133,-176.536,6.522,148.170
C06842=1232.104,280.114,-64.161,-176.534,6.524,148.169
C06843=1232.099,280.363,-64.188,-176.531,6.526,148.169
C06844=1232.095,280.612,-64.216,-176.529,6.528,148.169
C06845=1232.090,280.860,-64.245,-176.527,6.530,148.169
C06846=1232.086,281.108,-64.273,-176.525,6.532,148.169
C06847=1232.082,281.356,-64.301,-176.522,6.534,148.168
C06848=1232.077,281.605,-64.330,-176.519,6.537,148.168
C06849=1232.073,281.853,-64.357,-176.517,6.539,148.168
C06850=1232.069,282.102,-64.386,-176.515,6.541,148.168
C06851=1232.064,282.350,-64.414,-176.512,6.543,148.168
C06852=1232.060,282.599,-64.443,-176.510,6.545,148.168
C06853=1232.055,282.847,-64.470,-176.507,6.547,148.167
C06854=1232.052,283.095,-64.498,-176.505,6.549,148.167
C06855=1232.047,283.343,-64.528,-176.503,6.552,148.167
C06856=1232.043,283.591,-64.556,-176.500,6.554,148.167
C06857=1232.039,283.840,-64.584,-176.498,6.557,148.167
C06858=1232.034,284.088,-64.612,-176.495,6.559,148.167
C06859=1232.030,284.337,-64.641,-176.493,6.561,148.167
C06860=1232.025,284.585,-64.669,-176.491,6.563,148.167
C06861=1232.021,284.834,-64.697,-176.488,6.566,148.166
C06862=1232.016,285.082,-64.726,-176.486,6.568,148.166
C06863=1232.012,285.330,-64.754,-176.483,6.570,148.166
C06864=1232.007,285.578,-64.783,-176.481,6.572,148.166
C06865=1232.004,285.827,-64.811,-176.479,6.574,148.166
C06866=1231.999,286.075,-64.840,-176.476,6.576,148.166
C06867=1231.995,286.323,-64.868,-176.474,6.579,148.166
C06868=1231.990,286.572,-64.896,-176.471,6.581,148.165
C06869=1231.986,286.819,-64.925,-176.469,6.583,148.165
C06870=1231.982,287.068,-64.954,-176.467,6.586,148.165
C06871=1231.977,287.317,-64.982,-176.464,6.587,148.165
C06872=1231.973,287.565,-65.010,-176.462,6.590,148.165
C06873=1231.969,287.813,-65.040,-176.459,6.592,148.165
C06874=1231.964,288.061,-65.067,-176.457,6.595,148.165
C06875=1231.960,288.310,-65.096,-176.455,6.597,148.164
C06876=1231.955,288.559,-65.125,-176.452,6.599,148.164
C06877=1231.951,288.806,-65.153,-176.450,6.601,148.164
C06878=1231.947,289.055,-65.182,-176.448,6.603,148.164
C06879=1231.942,289.330,-65.214,-176.445,6.606,148.164
C06880=1231.937,289.603,-65.245,-176.442,6.609,148.164
C06881=1231.932,289.877,-65.277,-176.440,6.611,148.164
C06882=1231.927,290.151,-65.309,-176.437,6.614,148.164
C06883=1231.924,290.400,-65.337,-176.435,6.616,148.163
C06884=1231.919,290.647,-65.366,-176.432,6.618,148.163
C06885=1231.914,290.896,-65.395,-176.430,6.620,148.163
C06886=1231.911,291.144,-65.424,-176.428,6.622,148.163
C06887=1231.906,291.392,-65.452,-176.426,6.624,148.163
C06888=1231.901,291.641,-65.481,-176.423,6.628,148.163
C06889=1231.897,291.890,-65.510,-176.421,6.630,148.163
C06890=1231.893,292.137,-65.538,-176.418,6.632,148.162
C06891=1231.889,292.386,-65.568,-176.416,6.634,148.162
C06892=1231.884,292.635,-65.596,-176.414,6.636,148.162
C06893=1231.879,292.882,-65.625,-176.411,6.639,148.162
C06894=1231.876,293.131,-65.654,-176.409,6.641,148.162
C06895=1231.871,293.379,-65.683,-176.407,6.643,148.162
C06896=1231.867,293.628,-65.712,-176.405,6.646,148.162
C06897=1231.862,293.875,-65.741,-176.402,6.647,148.162
C06898=1231.858,294.124,-65.769,-176.399,6.650,148.162
C06899=1231.854,294.372,-65.799,-176.397,6.653,148.162
C06900=1231.849,294.620,-65.828,-176.395,6.655,148.161
C06901=1231.845,294.869,-65.856,-176.393,6.657,148.161
C06902=1231.841,295.117,-65.886,-176.390,6.660,148.161
C06903=1231.836,295.366,-65.915,-176.388,6.662,148.161
C06904=1231.832,295.613,-65.943,-176.385,6.664,148.161
C06905=1231.828,295.861,-65.972,-176.383,6.666,148.161
C06906=1231.824,296.110,-66.001,-176.381,6.668,148.161
C06907=1231.819,296.359,-66.031,-176.378,6.672,148.161
C06908=1231.815,296.606,-66.060,-176.376,6.673,148.160
C06909=1231.810,296.855,-66.088,-176.374,6.676,148.160
C06910=1231.806,297.103,-66.118,-176.372,6.678,148.160
C06911=1231.802,297.351,-66.147,-176.369,6.680,148.160
C06912=1231.798,297.600,-66.176,-176.367,6.683,148.160
C06913=1231.793,297.848,-66.205,-176.364,6.685,148.160
C06914=1231.789,298.096,-66.234,-176.362,6.687,148.160
C06915=1231.785,298.344,-66.264,-176.360,6.690,148.160
C06916=1231.780,298.593,-66.292,-176.357,6.693,148.160
C06917=1231.776,298.841,-66.322,-176.355,6.695,148.160
C06918=1231.771,299.089,-66.351,-176.353,6.697,148.160
C06919=1231.767,299.337,-66.380,-176.351,6.699,148.159
C06920=1231.763,299.586,-66.409,-176.348,6.701,148.159
C06921=1231.758,299.834,-66.438,-176.346,6.704,148.159
C06922=1231.754,300.083,-66.468,-176.344,6.706,148.159
C06923=1231.750,300.331,-66.497,-176.342,6.709,148.159
C06924=1231.745,300.579,-66.526,-176.339,6.711,148.159
C06925=1231.741,300.827,-66.556,-176.336,6.714,148.159
C06926=1231.737,301.076,-66.585,-176.334,6.716,148.159
C06927=1231.732,301.324,-66.614,-176.332,6.718,148.159
C06928=1231.728,301.572,-66.644,-176.330,6.720,148.159
C06929=1231.724,301.820,-66.673,-176.327,6.723,148.159
C06930=1231.719,302.068,-66.702,-176.325,6.725,148.159
C06931=1231.715,302.316,-66.732,-176.323,6.728,148.159
C06932=1231.711,302.565,-66.761,-176.321,6.730,148.158
C06933=1231.707,302.813,-66.790,-176.319,6.732,148.158
C06934=1231.703,303.061,-66.820,-176.316,6.735,148.158
C06935=1231.698,303.309,-66.849,-176.314,6.737,148.158
C06936=1231.694,303.558,-66.879,-176.312,6.739,148.158
C06937=1231.690,303.806,-66.908,-176.310,6.742,148.158
C06938=1231.685,304.053,-66.937,-176.306,6.744,148.158
C06939=1231.681,304.302,-66.967,-176.304,6.747,148.158
C06940=1231.677,304.550,-66.996,-176.302,6.749,148.158
C06941=1231.672,304.799,-67.026,-176.300,6.751,148.158
C06942=1231.668,305.047,-67.056,-176.297,6.754,148.158
C06943=1231.664,305.295,-67.085,-176.295,6.756,148.158
C06944=1231.659,305.543,-67.115,-176.293,6.759,148.158
C06945=1231.655,305.792,-67.144,-176.291,6.761,148.158
C06946=1231.651,306.040,-67.174,-176.289,6.764,148.158
C06947=1231.647,306.288,-67.203,-176.286,6.766,148.158
C06948=1231.642,306.537,-67.233,-176.284,6.768,148.158
C06949=1231.638,306.784,-67.263,-176.282,6.771,148.158
C06950=1231.634,307.033,-67.293,-176.280,6.774,148.158
C06951=1231.629,307.280,-67.322,-176.277,6.776,148.157
C06952=1231.625,307.529,-67.351,-176.275,6.778,148.157
C06953=1231.620,307.777,-67.381,-176.273,6.780,148.157
C06954=1231.616,308.025,-67.411,-176.270,6.783,148.157
C06955=1231.612,308.274,-67.440,-176.268,6.785,148.157
C06956=1231.608,308.521,-67.470,-176.266,6.788,148.157
C06957=1231.604,308.770,-67.500,-176.264,6.790,148.157
C06958=1231.599,309.018,-67.530,-176.261,6.793,148.157
C06959=1231.595,309.266,-67.559,-176.259,6.795,148.157
C06960=1231.591,309.514,-67.589,-176.257,6.797,148.157
C06961=1231.586,309.762,-67.619,-176.255,6.799,148.157
C06962=1231.582,310.011,-67.649,-176.252,6.803,148.157
C06963=1231.577,310.259,-67.678,-176.250,6.805,148.157
C06964=1231.574,310.507,-67.709,-176.248,6.807,148.157
C06965=1231.569,310.755,-67.739,-176.246,6.809,148.157
C06966=1231.564,311.004,-67.768,-176.243,6.812,148.157
C06967=1231.561,311.251,-67.798,-176.241,6.815,148.157
C06968=1231.556,311.500,-67.828,-176.240,6.817,148.157
C06969=1231.551,311.748,-67.858,-176.237,6.819,148.157
C06970=1231.548,311.996,-67.888,-176.235,6.822,148.157
C06971=1231.543,312.244,-67.917,-176.233,6.825,148.157
C06972=1231.538,312.493,-67.947,-176.231,6.827,148.157
C06973=1231.535,312.740,-67.978,-176.228,6.830,148.157
C06974=1231.531,312.989,-68.007,-176.226,6.832,148.157
C06975=1231.526,313.237,-68.038,-176.224,6.834,148.157
C06976=1231.522,313.485,-68.068,-176.222,6.837,148.156
C06977=1231.518,313.733,-68.098,-176.219,6.840,148.157
C06978=1231.513,313.982,-68.128,-176.217,6.842,148.156
C06979=1231.509,314.230,-68.157,-176.215,6.844,148.156
C06980=1231.505,314.478,-68.188,-176.213,6.846,148.156
C06981=1231.500,314.726,-68.218,-176.210,6.849,148.156
C06982=1231.497,314.974,-68.248,-176.208,6.852,148.157
C06983=1231.491,315.250,-68.281,-176.206,6.855,148.157
C06984=1231.487,315.525,-68.315,-176.204,6.857,148.156
C06985=1231.482,315.801,-68.348,-176.201,6.860,148.156
C06986=1231.478,316.077,-68.382,-176.199,6.862,148.156
C06987=1231.473,316.325,-68.412,-176.196,6.866,148.156
C06988=1231.469,316.573,-68.442,-176.194,6.868,148.156
C06989=1231.464,316.821,-68.473,-176.192,6.870,148.156
C06990=1231.460,317.069,-68.502,-176.189,6.873,148.156
C06991=1231.456,317.317,-68.533,-176.187,6.875,148.156
C06992=1231.451,317.566,-68.562,-176.186,6.878,148.156
C06993=1231.447,317.814,-68.594,-176.184,6.880,148.156
C06994=1231.443,318.062,-68.624,-176.181,6.883,148.156
C06995=1231.439,318.310,-68.654,-176.179,6.885,148.156
C06996=1231.435,318.558,-68.684,-176.177,6.888,148.156
C06997=1231.430,318.806,-68.715,-176.175,6.890,148.156
C06998=1231.426,319.054,-68.744,-176.173,6.893,148.157
C06999=1231.422,319.303,-68.775,-176.170,6.895,148.156
C07000=1231.418,319.551,-68.806,-176.168,6.898,148.156
C07001=1231.413,319.799,-68.836,-176.166,6.900,148.156
C07002=1231.409,320.047,-68.866,-176.164,6.903,148.156
C07003=1231.405,320.295,-68.896,-176.162,6.905,148.157
C07004=1231.401,320.542,-68.927,-176.160,6.908,148.157
C07005=1231.396,320.792,-68.957,-176.157,6.911,148.157
C07006=1231.392,321.040,-68.988,-176.155,6.913,148.156
C07007=1231.388,321.287,-69.018,-176.154,6.915,148.157
C07008=1231.383,321.535,-69.049,-176.151,6.918,148.157
C07009=1231.379,321.784,-69.078,-176.149,6.921,148.157
C07010=1231.375,322.032,-69.109,-176.147,6.923,148.157
C07011=1231.370,322.280,-69.140,-176.145,6.926,148.157
C07012=1231.367,322.528,-69.170,-176.143,6.928,148.157
C07013=1231.362,322.776,-69.201,-176.140,6.931,148.157
C07014=1231.359,323.024,-69.232,-176.138,6.933,148.157
C07015=1231.354,323.273,-69.262,-176.137,6.936,148.157
C07016=1231.349,323.521,-69.292,-176.134,6.939,148.157
C07017=1231.345,323.768,-69.323,-176.132,6.941,148.157
C07018=1231.341,324.016,-69.353,-176.130,6.943,148.157
C07019=1231.337,324.265,-69.384,-176.128,6.946,148.157
C07020=1231.333,324.513,-69.415,-176.125,6.949,148.157
C07021=1231.328,324.761,-69.445,-176.123,6.951,148.157
C07022=1231.324,325.009,-69.477,-176.122,6.953,148.157
C07023=1231.320,325.257,-69.507,-176.120,6.956,148.157
C07024=1231.316,325.505,-69.537,-176.117,6.959,148.157
C07025=1231.311,325.753,-69.568,-176.115,6.961,148.157
C07026=1231.307,326.001,-69.599,-176.113,6.963,148.157
C07027=1231.303,326.249,-69.630,-176.111,6.967,148.157
C07028=1231.299,326.497,-69.660,-176.109,6.969,148.157
C07029=1231.294,326.745,-69.691,-176.107,6.971,148.157
C07030=1231.290,326.994,-69.722,-176.105,6.974,148.157
C07031=1231.286,327.241,-69.752,-176.103,6.977,148.157
C07032=1231.281,327.489,-69.783,-176.101,6.979,148.157
C07033=1231.277,327.738,-69.814,-176.099,6.982,148.158
C07034=1231.273,327.986,-69.845,-176.097,6.984,148.158
C07035=1231.269,328.234,-69.875,-176.095,6.987,148.158
C07036=1231.265,328.482,-69.906,-176.093,6.990,148.158
C07037=1231.260,328.730,-69.937,-176.090,6.992,148.158
C07038=1231.256,328.978,-69.968,-176.088,6.995,148.158
C07039=1231.252,329.226,-70.000,-176.086,6.997,148.158
C07040=1231.247,329.474,-70.030,-176.085,7.000,148.158
C07041=1231.244,329.722,-70.061,-176.082,7.002,148.158
C07042=1231.239,329.970,-70.092,-176.080,7.005,148.158
C07043=1231.235,330.218,-70.123,-176.078,7.008,148.158
C07044=1231.230,330.466,-70.153,-176.076,7.010,148.158
C07045=1231.227,330.714,-70.185,-176.075,7.012,148.158
C07046=1231.222,330.962,-70.216,-176.072,7.016,148.158
C07047=1231.218,331.210,-70.246,-176.070,7.018,148.159
C07048=1231.214,331.459,-70.277,-176.068,7.020,148.159
C07049=1231.209,331.707,-70.308,-176.067,7.023,148.159
C07050=1231.205,331.954,-70.339,-176.064,7.026,148.159
C07051=1231.201,332.203,-70.371,-176.062,7.028,148.159
C07052=1231.197,332.451,-70.401,-176.060,7.031,148.159
C07053=1231.192,332.699,-70.432,-176.058,7.034,148.159
C07054=1231.188,332.947,-70.464,-176.056,7.036,148.159
C07055=1231.184,333.195,-70.495,-176.054,7.039,148.159
C07056=1231.180,333.443,-70.526,-176.052,7.041,148.159
C07057=1231.175,333.691,-70.557,-176.050,7.044,148.159
C07058=1231.171,333.939,-70.588,-176.048,7.047,148.159
C07059=1231.167,334.187,-70.619,-176.046,7.049,148.160
C07060=1231.163,334.434,-70.650,-176.044,7.051,148.160
C07061=1231.159,334.683,-70.681,-176.042,7.055,148.160
C07062=1231.154,334.931,-70.712,-176.040,7.057,148.160
C07063=1231.151,335.179,-70.744,-176.038,7.059,148.160
C07064=1231.146,335.427,-70.775,-176.037,7.062,148.160
C07065=1231.142,335.675,-70.806,-176.034,7.065,148.160
C07066=1231.138,335.923,-70.837,-176.032,7.068,148.160
C07067=1231.133,336.170,-70.869,-176.031,7.070,148.160
C07068=1231.129,336.419,-70.900,-176.029,7.072,148.160
C07069=1231.125,336.667,-70.931,-176.027,7.076,148.161
C07070=1231.121,336.915,-70.962,-176.024,7.078,148.161
C07071=1231.117,337.163,-70.993,-176.023,7.081,148.161
C07072=1231.112,337.411,-71.026,-176.021,7.083,148.161
C07073=1231.107,337.659,-71.056,-176.019,7.086,148.161
C07074=1231.104,337.907,-71.088,-176.017,7.089,148.161
C07075=1231.099,338.155,-71.119,-176.015,7.091,148.161
C07076=1231.095,338.403,-71.151,-176.013,7.093,148.161
C07077=1231.091,338.651,-71.182,-176.011,7.097,148.162
C07078=1231.087,338.899,-71.213,-176.009,7.099,148.162
C07079=1231.083,339.146,-71.245,-176.007,7.102,148.162
C07080=1231.079,339.395,-71.276,-176.006,7.104,148.162
C07081=1231.075,339.642,-71.308,-176.004,7.107,148.162
C07082=1231.071,339.891,-71.339,-176.001,7.110,148.162
C07083=1231.066,340.138,-71.370,-176.000,7.112,148.162
C07084=1231.062,340.387,-71.403,-175.998,7.115,148.162
C07085=1231.057,340.635,-71.433,-175.996,7.118,148.162
C07086=1231.053,340.883,-71.465,-175.994,7.120,148.163
C07087=1231.048,341.160,-71.500,-175.992,7.123,148.163
C07088=1231.044,341.438,-71.535,-175.990,7.126,148.163
C07089=1231.040,341.715,-71.571,-175.988,7.129,148.163
C07090=1231.034,341.993,-71.605,-175.986,7.132,148.163
C07091=1231.031,342.241,-71.637,-175.984,7.134,148.163
C07092=1231.026,342.488,-71.669,-175.982,7.137,148.163
C07093=1231.022,342.737,-71.701,-175.980,7.140,148.164
C07094=1231.018,342.985,-71.732,-175.978,7.143,148.164
C07095=1231.014,343.232,-71.764,-175.977,7.145,148.164
C07096=1231.009,343.481,-71.796,-175.975,7.148,148.164
C07097=1231.005,343.729,-71.827,-175.972,7.151,148.164
C07098=1231.001,343.977,-71.859,-175.971,7.153,148.164
C07099=1230.996,344.224,-71.890,-175.969,7.156,148.165
C07100=1230.993,344.472,-71.922,-175.967,7.159,148.165
C07101=1230.988,344.721,-71.954,-175.965,7.162,148.165
C07102=1230.984,344.968,-71.985,-175.963,7.164,148.165
C07103=1230.980,345.216,-72.017,-175.962,7.166,148.165
C07104=1230.975,345.464,-72.049,-175.960,7.169,148.165
C07105=1230.971,345.712,-72.081,-175.958,7.172,148.165
C07106=1230.967,345.959,-72.113,-175.956,7.175,148.166
C07107=1230.963,346.208,-72.144,-175.955,7.177,148.166
C07108=1230.959,346.457,-72.176,-175.953,7.180,148.166
C07109=1230.954,346.704,-72.208,-175.951,7.182,148.166
C07110=1230.950,346.952,-72.240,-175.949,7.185,148.166
C07111=1230.946,347.200,-72.272,-175.947,7.188,148.166
C07112=1230.942,347.448,-72.303,-175.946,7.191,148.167
C07113=1230.938,347.696,-72.335,-175.944,7.193,148.167
C07114=1230.933,347.943,-72.367,-175.942,7.196,148.167
C07115=1230.929,348.191,-72.399,-175.940,7.199,148.167
C07116=1230.926,348.439,-72.431,-175.939,7.202,148.167
C07117=1230.921,348.687,-72.463,-175.937,7.204,148.168
C07118=1230.917,348.935,-72.495,-175.935,7.207,148.168
C07119=1230.913,349.184,-72.526,-175.934,7.209,148.168
C07120=1230.908,349.431,-72.558,-175.931,7.212,148.168
C07121=1230.904,349.679,-72.590,-175.930,7.215,148.168
C07122=1230.900,349.927,-72.622,-175.928,7.218,148.169
C07123=1230.896,350.174,-72.655,-175.927,7.220,148.169
C07124=1230.892,350.422,-72.687,-175.925,7.223,148.169
C07125=1230.887,350.671,-72.719,-175.923,7.226,148.169
C07126=1230.883,350.918,-72.750,-175.921,7.228,148.169
C07127=1230.879,351.166,-72.782,-175.920,7.231,148.169
C07128=1230.875,351.415,-72.815,-175.918,7.234,148.170
C07129=1230.871,351.662,-72.846,-175.916,7.236,148.170
C07130=1230.866,351.910,-72.879,-175.915,7.239,148.170
C07131=1230.863,352.158,-72.910,-175.913,7.242,148.170
C07132=1230.858,352.406,-72.943,-175.911,7.245,148.170
C07133=1230.854,352.654,-72.974,-175.909,7.247,148.171
C07134=1230.849,352.902,-73.007,-175.908,7.250,148.171
C07135=1230.846,353.150,-73.039,-175.906,7.252,148.171
C07136=1230.841,353.397,-73.071,-175.904,7.255,148.171
C07137=1230.837,353.645,-73.103,-175.902,7.258,148.171
C07138=1230.833,353.894,-73.136,-175.901,7.261,148.172
C07139=1230.828,354.141,-73.167,-175.899,7.263,148.172
C07140=1230.824,354.389,-73.200,-175.897,7.266,148.172
C07141=1230.821,354.637,-73.232,-175.896,7.268,148.172
C07142=1230.816,354.885,-73.265,-175.895,7.271,148.173
C07143=1230.812,355.133,-73.296,-175.892,7.274,148.173
C07144=1230.807,355.381,-73.329,-175.891,7.277,148.173
C07145=1230.804,355.628,-73.361,-175.889,7.279,148.173
C07146=1230.800,355.877,-73.394,-175.888,7.282,148.173
C07147=1230.795,356.124,-73.425,-175.886,7.284,148.174
C07148=1230.791,356.372,-73.458,-175.884,7.287,148.174
C07149=1230.787,356.620,-73.490,-175.883,7.290,148.174
C07150=1230.783,356.868,-73.523,-175.881,7.293,148.174
C07151=1230.779,357.115,-73.554,-175.879,7.296,148.175
C07152=1230.775,357.363,-73.587,-175.878,7.298,148.175
C07153=1230.770,357.612,-73.620,-175.876,7.301,148.175
C07154=1230.766,357.860,-73.651,-175.875,7.304,148.175
C07155=1230.762,358.107,-73.685,-175.873,7.306,148.176
C07156=1230.758,358.355,-73.716,-175.872,7.309,148.176
C07157=1230.753,358.603,-73.749,-175.870,7.311,148.176
C07158=1230.749,358.851,-73.782,-175.868,7.315,148.176
C07159=1230.746,359.099,-73.814,-175.867,7.317,148.177
C07160=1230.741,359.347,-73.846,-175.865,7.320,148.177
C07161=1230.737,359.594,-73.878,-175.863,7.322,148.177
C07162=1230.733,359.842,-73.911,-175.862,7.325,148.177
C07163=1230.729,360.090,-73.944,-175.861,7.328,148.177
C07164=1230.725,360.338,-73.976,-175.859,7.330,148.178
C07165=1230.720,360.586,-74.008,-175.857,7.333,148.178
C07166=1230.716,360.834,-74.041,-175.856,7.336,148.178
C07167=1230.712,361.081,-74.073,-175.855,7.338,148.178
C07168=1230.708,361.329,-74.106,-175.853,7.342,148.179
C07169=1230.703,361.577,-74.138,-175.851,7.344,148.179
C07170=1230.700,361.825,-74.171,-175.850,7.347,148.179
C07171=1230.696,362.073,-74.203,-175.848,7.350,148.179
C07172=1230.691,362.321,-74.236,-175.847,7.352,148.180
C07173=1230.687,362.568,-74.268,-175.845,7.355,148.180
C07174=1230.683,362.816,-74.301,-175.844,7.357,148.180
C07175=1230.679,363.064,-74.334,-175.843,7.360,148.181
C07176=1230.674,363.312,-74.367,-175.841,7.363,148.181
C07177=1230.671,363.560,-74.399,-175.840,7.366,148.181
C07178=1230.667,363.808,-74.432,-175.838,7.368,148.181
C07179=1230.662,364.056,-74.465,-175.837,7.371,148.182
C07180=1230.659,364.304,-74.497,-175.835,7.373,148.182
C07181=1230.654,364.551,-74.529,-175.834,7.376,148.182
C07182=1230.650,364.799,-74.562,-175.833,7.379,148.183
C07183=1230.645,365.047,-74.595,-175.830,7.382,148.183
C07184=1230.642,365.294,-74.628,-175.829,7.385,148.183
C07185=1230.638,365.543,-74.660,-175.828,7.388,148.183
C07186=1230.633,365.790,-74.693,-175.826,7.390,148.184
C07187=1230.629,366.038,-74.726,-175.825,7.393,148.184
C07188=1230.625,366.286,-74.759,-175.823,7.395,148.184
C07189=1230.621,366.534,-74.791,-175.822,7.398,148.185
C07190=1230.617,366.781,-74.825,-175.820,7.401,148.185
C07191=1230.612,367.061,-74.861,-175.819,7.404,148.185
C07192=1230.607,367.341,-74.899,-175.817,7.407,148.185
C07193=1230.603,367.620,-74.935,-175.816,7.410,148.186
C07194=1230.598,367.899,-74.972,-175.815,7.413,148.186
C07195=1230.594,368.147,-75.005,-175.813,7.415,148.186
C07196=1230.590,368.395,-75.038,-175.812,7.418,148.187
C07197=1230.585,368.643,-75.071,-175.810,7.421,148.187
C07198=1230.582,368.891,-75.103,-175.809,7.423,148.187
C07199=1230.578,369.138,-75.136,-175.808,7.426,148.188
C07200=1230.573,369.386,-75.170,-175.806,7.429,148.188
C07201=1230.569,369.634,-75.203,-175.805,7.432,148.188
C07202=1230.565,369.882,-75.235,-175.804,7.434,148.189
C07203=1230.561,370.130,-75.268,-175.802,7.437,148.189
C07204=1230.557,370.378,-75.301,-175.801,7.439,148.189
C07205=1230.552,370.625,-75.335,-175.800,7.442,148.190
C07206=1230.549,370.873,-75.367,-175.799,7.445,148.190
C07207=1230.545,371.121,-75.400,-175.797,7.448,148.190
C07208=1230.540,371.369,-75.433,-175.796,7.450,148.191
C07209=1230.536,371.616,-75.466,-175.794,7.453,148.191
C07210=1230.532,371.864,-75.499,-175.793,7.456,148.191
C07211=1230.528,372.112,-75.532,-175.792,7.459,148.192
C07212=1230.524,372.360,-75.565,-175.790,7.461,148.192
C07213=1230.520,372.607,-75.599,-175.790,7.463,148.192
C07214=1230.515,372.856,-75.631,-175.788,7.466,148.192
C07215=1230.511,373.103,-75.664,-175.787,7.469,148.193
C07216=1230.507,373.351,-75.697,-175.786,7.471,148.193
C07217=1230.503,373.599,-75.730,-175.784,7.474,148.193
C07218=1230.499,373.847,-75.764,-175.783,7.477,148.194
C07219=1230.495,374.094,-75.797,-175.782,7.480,148.194
C07220=1230.491,374.342,-75.830,-175.780,7.482,148.194
C07221=1230.486,374.590,-75.863,-175.779,7.485,148.195
C07222=1230.482,374.838,-75.896,-175.779,7.487,148.195
C07223=1230.478,375.085,-75.929,-175.777,7.490,148.195
C07224=1230.474,375.333,-75.963,-175.776,7.493,148.196
C07225=1230.470,375.581,-75.996,-175.775,7.495,148.196
C07226=1230.466,375.829,-76.029,-175.774,7.498,148.197
C07227=1230.462,376.076,-76.062,-175.772,7.501,148.197
C07228=1230.457,376.324,-76.095,-175.771,7.504,148.197
C07229=1230.453,376.572,-76.128,-175.770,7.505,148.197
C07230=1230.449,376.819,-76.161,-175.769,7.508,148.198
C07231=1230.445,377.067,-76.195,-175.768,7.511,148.198
C07232=1230.441,377.315,-76.228,-175.766,7.514,148.198
C07233=1230.437,377.563,-76.261,-175.765,7.517,148.199
C07234=1230.433,377.810,-76.294,-175.764,7.519,148.199
C07235=1230.428,378.058,-76.327,-175.763,7.521,148.200
C07236=1230.424,378.306,-76.360,-175.762,7.524,148.200
C07237=1230.420,378.554,-76.394,-175.760,7.527,148.200
C07238=1230.417,378.801,-76.428,-175.759,7.529,148.201
C07239=1230.413,379.049,-76.461,-175.758,7.532,148.201
C07240=1230.409,379.297,-76.494,-175.758,7.534,148.201
C07241=1230.405,379.545,-76.527,-175.756,7.537,148.202
C07242=1230.400,379.793,-76.561,-175.755,7.540,148.202
C07243=1230.396,380.040,-76.594,-175.754,7.543,148.203
C07244=1230.391,380.288,-76.627,-175.753,7.546,148.203
C07245=1230.387,380.536,-76.660,-175.752,7.547,148.203
C07246=1230.383,380.783,-76.694,-175.751,7.550,148.203
C07247=1230.379,381.031,-76.727,-175.749,7.553,148.204
C07248=1230.375,381.278,-76.761,-175.748,7.556,148.204
C07249=1230.371,381.526,-76.794,-175.748,7.558,148.205
C07250=1230.367,381.775,-76.828,-175.747,7.561,148.205
C07251=1230.363,382.022,-76.862,-175.745,7.563,148.205
C07252=1230.359,382.270,-76.895,-175.744,7.566,148.206
C07253=1230.355,382.517,-76.928,-175.744,7.568,148.206
C07254=1230.350,382.765,-76.961,-175.742,7.571,148.207
C07255=1230.346,383.013,-76.994,-175.741,7.574,148.207
C07256=1230.342,383.260,-77.029,-175.741,7.576,148.207
C07257=1230.338,383.508,-77.062,-175.739,7.579,148.208
C07258=1230.333,383.756,-77.095,-175.738,7.581,148.208
C07259=1230.330,384.004,-77.129,-175.738,7.583,148.208
C07260=1230.326,384.251,-77.163,-175.737,7.586,148.209
C07261=1230.322,384.499,-77.196,-175.735,7.589,148.209
C07262=1230.317,384.747,-77.229,-175.734,7.592,148.210
C07263=1230.313,384.994,-77.263,-175.734,7.594,148.210
C07264=1230.309,385.242,-77.297,-175.732,7.597,148.210
C07265=1230.305,385.490,-77.330,-175.731,7.600,148.211
C07266=1230.302,385.737,-77.364,-175.731,7.602,148.211
C07267=1230.297,385.985,-77.398,-175.729,7.604,148.212
C07268=1230.293,386.233,-77.431,-175.728,7.607,148.212
C07269=1230.289,386.480,-77.465,-175.728,7.609,148.212
C07270=1230.285,386.728,-77.498,-175.726,7.612,148.213
C07271=1230.280,386.976,-77.532,-175.725,7.615,148.213
C07272=1230.277,387.224,-77.566,-175.725,7.617,148.213
C07273=1230.273,387.472,-77.599,-175.724,7.620,148.214
C07274=1230.268,387.719,-77.632,-175.723,7.622,148.214
C07275=1230.264,387.967,-77.667,-175.722,7.624,148.215
C07276=1230.260,388.214,-77.700,-175.721,7.627,148.215
C07277=1230.256,388.462,-77.734,-175.720,7.629,148.215
C07278=1230.252,388.710,-77.767,-175.719,7.632,148.216
C07279=1230.247,388.958,-77.801,-175.718,7.634,148.216
C07280=1230.244,389.205,-77.835,-175.717,7.637,148.216
C07281=1230.239,389.453,-77.868,-175.716,7.640,148.217
C07282=1230.235,389.700,-77.902,-175.715,7.642,148.217
C07283=1230.231,389.949,-77.936,-175.714,7.645,148.218
C07284=1230.228,390.196,-77.970,-175.713,7.646,148.218
C07285=1230.223,390.444,-78.003,-175.713,7.650,148.219
C07286=1230.219,390.691,-78.037,-175.712,7.652,148.219
C07287=1230.215,390.939,-78.071,-175.711,7.654,148.219
C07288=1230.211,391.187,-78.105,-175.710,7.657,148.220
C07289=1230.207,391.435,-78.139,-175.709,7.659,148.220
C07290=1230.203,391.682,-78.172,-175.708,7.662,148.220
C07291=1230.199,391.929,-78.206,-175.707,7.664,148.221
C07292=1230.195,392.178,-78.240,-175.706,7.667,148.221
C07293=1230.191,392.425,-78.274,-175.706,7.669,148.222
C07294=1230.187,392.672,-78.307,-175.705,7.672,148.222
C07295=1230.181,392.955,-78.346,-175.704,7.675,148.223
C07296=1230.177,393.235,-78.385,-175.702,7.678,148.223
C07297=1230.172,393.517,-78.423,-175.702,7.680,148.223
C07298=1230.168,393.798,-78.461,-175.701,7.683,148.224
C07299=1230.163,394.046,-78.494,-175.700,7.686,148.224
C07300=1230.159,394.294,-78.529,-175.699,7.688,148.225
C07301=1230.156,394.541,-78.563,-175.698,7.690,148.225
C07302=1230.151,394.788,-78.596,-175.698,7.692,148.225
C07303=1230.147,395.036,-78.631,-175.697,7.695,148.226
C07304=1230.143,395.284,-78.664,-175.696,7.697,148.226
C07305=1230.139,395.532,-78.699,-175.695,7.700,148.227
C07306=1230.135,395.779,-78.733,-175.694,7.702,148.227
C07307=1230.131,396.027,-78.766,-175.693,7.705,148.227
